// ---- VISUs/Parameter/Recipe/MOffset_1.TcVIS
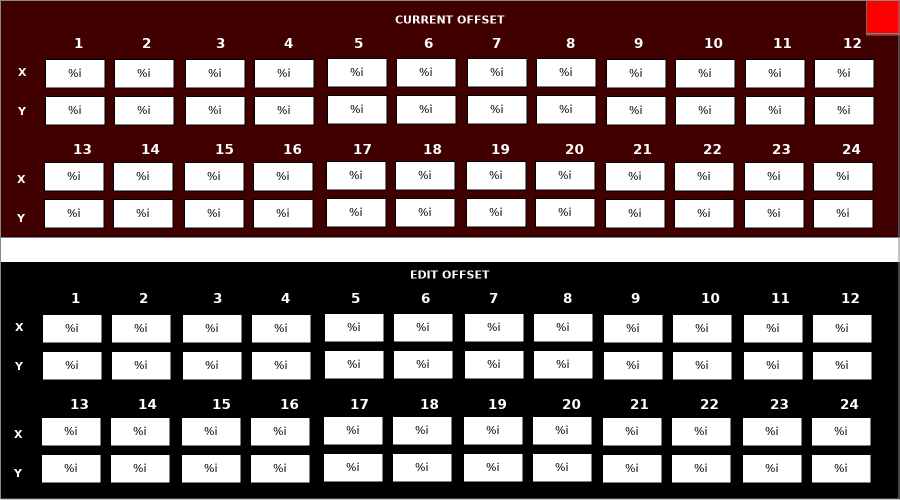
VISUALIZATION MOffset_1  // 900x500
    RoundedRectangle (0,0 900x237)
    Label (0,0 900x40), "CURRENT OFFSET"
    Label (15,55 25x35), "X"
    RoundedRectangle (45,59 60x29), "%i", text variable: Status_GVL.RecipeLine[1].OffsetPattern.Offset_X[1]
    Label (71,26 25x35), "1"
    RoundedRectangle (114,59 60x29), "%i", text variable: Status_GVL.RecipeLine[1].OffsetPattern.Offset_X[2]
    Label (139,26 25x35), "2"
    RoundedRectangle (185,59 60x29), "%i", text variable: Status_GVL.RecipeLine[1].OffsetPattern.Offset_X[3]
    RoundedRectangle (254,59 60x29), "%i", text variable: Status_GVL.RecipeLine[1].OffsetPattern.Offset_X[4]
    Label (15,94 25x35), "Y"
    RoundedRectangle (327,58 60x29), "%i", text variable: Status_GVL.RecipeLine[1].OffsetPattern.Offset_X[5]
    RoundedRectangle (396,58 60x29), "%i", text variable: Status_GVL.RecipeLine[1].OffsetPattern.Offset_X[6]
    RoundedRectangle (467,58 60x29), "%i", text variable: Status_GVL.RecipeLine[1].OffsetPattern.Offset_X[7]
    RoundedRectangle (536,58 60x29), "%i", text variable: Status_GVL.RecipeLine[1].OffsetPattern.Offset_X[8]
    RoundedRectangle (606,59 60x29), "%i", text variable: Status_GVL.RecipeLine[1].OffsetPattern.Offset_X[9]
    RoundedRectangle (675,59 60x29), "%i", text variable: Status_GVL.RecipeLine[1].OffsetPattern.Offset_X[10]
    Label (213,26 25x35), "3"
    Label (281,26 25x35), "4"
    Label (351,26 25x35), "5"
    Label (421,26 25x35), "6"
    Label (489,26 25x35), "7"
    Label (563,26 25x35), "8"
    Label (631,26 25x35), "9"
    Label (701,26 25x35), "10"
    RoundedRectangle (45,96 60x29), "%i", text variable: Status_GVL.RecipeLine[1].OffsetPattern.Offset_Y[1]
    RoundedRectangle (114,96 60x29), "%i", text variable: Status_GVL.RecipeLine[1].OffsetPattern.Offset_Y[2]
    RoundedRectangle (185,96 60x29), "%i", text variable: Status_GVL.RecipeLine[1].OffsetPattern.Offset_Y[3]
    RoundedRectangle (254,96 60x29), "%i", text variable: Status_GVL.RecipeLine[1].OffsetPattern.Offset_Y[4]
    RoundedRectangle (327,95 60x29), "%i", text variable: Status_GVL.RecipeLine[1].OffsetPattern.Offset_Y[5]
    RoundedRectangle (396,95 60x29), "%i", text variable: Status_GVL.RecipeLine[1].OffsetPattern.Offset_Y[6]
    RoundedRectangle (467,95 60x29), "%i", text variable: Status_GVL.RecipeLine[1].OffsetPattern.Offset_Y[7]
    RoundedRectangle (536,95 60x29), "%i", text variable: Status_GVL.RecipeLine[1].OffsetPattern.Offset_Y[8]
    RoundedRectangle (606,96 60x29), "%i", text variable: Status_GVL.RecipeLine[1].OffsetPattern.Offset_Y[9]
    RoundedRectangle (675,96 60x29), "%i", text variable: Status_GVL.RecipeLine[1].OffsetPattern.Offset_Y[10]
    Label (14,162 25x35), "X"
    RoundedRectangle (44,162 60x29), "%i", text variable: Status_GVL.RecipeLine[1].OffsetPattern.Offset_X[13]
    RoundedRectangle (113,162 60x29), "%i", text variable: Status_GVL.RecipeLine[1].OffsetPattern.Offset_X[14]
    RoundedRectangle (184,162 60x29), "%i", text variable: Status_GVL.RecipeLine[1].OffsetPattern.Offset_X[15]
    RoundedRectangle (253,162 60x29), "%i", text variable: Status_GVL.RecipeLine[1].OffsetPattern.Offset_X[16]
    Label (14,201 25x35), "Y"
    RoundedRectangle (326,161 60x29), "%i", text variable: Status_GVL.RecipeLine[1].OffsetPattern.Offset_X[17]
    RoundedRectangle (395,161 60x29), "%i", text variable: Status_GVL.RecipeLine[1].OffsetPattern.Offset_X[18]
    RoundedRectangle (466,161 60x29), "%i", text variable: Status_GVL.RecipeLine[1].OffsetPattern.Offset_X[19]
    RoundedRectangle (535,161 60x29), "%i", text variable: Status_GVL.RecipeLine[1].OffsetPattern.Offset_X[20]
    RoundedRectangle (605,162 60x29), "%i", text variable: Status_GVL.RecipeLine[1].OffsetPattern.Offset_X[21]
    RoundedRectangle (674,162 60x29), "%i", text variable: Status_GVL.RecipeLine[1].OffsetPattern.Offset_X[22]
    RoundedRectangle (44,199 60x29), "%i", text variable: Status_GVL.RecipeLine[1].OffsetPattern.Offset_Y[13]
    RoundedRectangle (113,199 60x29), "%i", text variable: Status_GVL.RecipeLine[1].OffsetPattern.Offset_Y[14]
    RoundedRectangle (184,199 60x29), "%i", text variable: Status_GVL.RecipeLine[1].OffsetPattern.Offset_Y[15]
    RoundedRectangle (253,199 60x29), "%i", text variable: Status_GVL.RecipeLine[1].OffsetPattern.Offset_Y[16]
    RoundedRectangle (326,198 60x29), "%i", text variable: Status_GVL.RecipeLine[1].OffsetPattern.Offset_Y[17]
    RoundedRectangle (395,198 60x29), "%i", text variable: Status_GVL.RecipeLine[1].OffsetPattern.Offset_Y[18]
    RoundedRectangle (466,198 60x29), "%i", text variable: Status_GVL.RecipeLine[1].OffsetPattern.Offset_Y[19]
    RoundedRectangle (535,198 60x29), "%i", text variable: Status_GVL.RecipeLine[1].OffsetPattern.Offset_Y[20]
    RoundedRectangle (605,199 60x29), "%i", text variable: Status_GVL.RecipeLine[1].OffsetPattern.Offset_Y[21]
    RoundedRectangle (674,199 60x29), "%i", text variable: Status_GVL.RecipeLine[1].OffsetPattern.Offset_Y[22]
    Label (70,132 25x35), "13"
    Label (138,132 25x35), "14"
    Label (212,132 25x35), "15"
    Label (280,132 25x35), "16"
    Label (350,132 25x35), "17"
    Label (420,132 25x35), "18"
    Label (488,132 25x35), "19"
    Label (562,132 25x35), "20"
    Label (630,132 25x35), "21"
    Label (700,132 25x35), "22"
    RoundedRectangle (0,262 900x237)
    Label (0,255 900x40), "EDIT OFFSET"
    Label (12,310 25x35), "X"
    RoundedRectangle (42,314 60x29), "%i", text variable: HMI_GVL.arRecipeHMI[1].OffsetPattern.Offset_X[1], input disabled if: Status_GVL.StsEdit[1]
        OnMouseClick: write the text variable via Default
    Label (68,281 25x35), "1"
    RoundedRectangle (111,314 60x29), "%i", text variable: HMI_GVL.arRecipeHMI[1].OffsetPattern.Offset_X[2], input disabled if: Status_GVL.StsEdit[1]
        OnMouseClick: write the text variable via Default
    Label (136,281 25x35), "2"
    RoundedRectangle (182,314 60x29), "%i", text variable: HMI_GVL.arRecipeHMI[1].OffsetPattern.Offset_X[3], input disabled if: Status_GVL.StsEdit[1]
        OnMouseClick: write the text variable via Default
    RoundedRectangle (251,314 60x29), "%i", text variable: HMI_GVL.arRecipeHMI[1].OffsetPattern.Offset_X[4], input disabled if: Status_GVL.StsEdit[1]
        OnMouseClick: write the text variable via Default
    Label (12,349 25x35), "Y"
    RoundedRectangle (324,313 60x29), "%i", text variable: HMI_GVL.arRecipeHMI[1].OffsetPattern.Offset_X[5], input disabled if: Status_GVL.StsEdit[1]
        OnMouseClick: write the text variable via Default
    RoundedRectangle (393,313 60x29), "%i", text variable: HMI_GVL.arRecipeHMI[1].OffsetPattern.Offset_X[6], input disabled if: Status_GVL.StsEdit[1]
        OnMouseClick: write the text variable via Default
    RoundedRectangle (464,313 60x29), "%i", text variable: HMI_GVL.arRecipeHMI[1].OffsetPattern.Offset_X[7], input disabled if: Status_GVL.StsEdit[1]
        OnMouseClick: write the text variable via Default
    RoundedRectangle (533,313 60x29), "%i", text variable: HMI_GVL.arRecipeHMI[1].OffsetPattern.Offset_X[8], input disabled if: Status_GVL.StsEdit[1]
        OnMouseClick: write the text variable via Default
    RoundedRectangle (603,314 60x29), "%i", text variable: HMI_GVL.arRecipeHMI[1].OffsetPattern.Offset_X[9], input disabled if: Status_GVL.StsEdit[1]
        OnMouseClick: write the text variable via Default
    RoundedRectangle (672,314 60x29), "%i", text variable: HMI_GVL.arRecipeHMI[1].OffsetPattern.Offset_X[10], input disabled if: Status_GVL.StsEdit[1]
        OnMouseClick: write the text variable via Default
    Label (210,281 25x35), "3"
    Label (278,281 25x35), "4"
    Label (348,281 25x35), "5"
    Label (418,281 25x35), "6"
    Label (486,281 25x35), "7"
    Label (560,281 25x35), "8"
    Label (628,281 25x35), "9"
    Label (698,281 25x35), "10"
    RoundedRectangle (42,351 60x29), "%i", text variable: HMI_GVL.arRecipeHMI[1].OffsetPattern.Offset_Y[1], input disabled if: Status_GVL.StsEdit[1]
        OnMouseClick: write the text variable via Default
    RoundedRectangle (111,351 60x29), "%i", text variable: HMI_GVL.arRecipeHMI[1].OffsetPattern.Offset_Y[2], input disabled if: Status_GVL.StsEdit[1]
        OnMouseClick: write the text variable via Default
    RoundedRectangle (182,351 60x29), "%i", text variable: HMI_GVL.arRecipeHMI[1].OffsetPattern.Offset_Y[3], input disabled if: Status_GVL.StsEdit[1]
        OnMouseClick: write the text variable via Default
    RoundedRectangle (251,351 60x29), "%i", text variable: HMI_GVL.arRecipeHMI[1].OffsetPattern.Offset_Y[4], input disabled if: Status_GVL.StsEdit[1]
        OnMouseClick: write the text variable via Default
    RoundedRectangle (324,350 60x29), "%i", text variable: HMI_GVL.arRecipeHMI[1].OffsetPattern.Offset_Y[5], input disabled if: Status_GVL.StsEdit[1]
        OnMouseClick: write the text variable via Default
    RoundedRectangle (393,350 60x29), "%i", text variable: HMI_GVL.arRecipeHMI[1].OffsetPattern.Offset_Y[6], input disabled if: Status_GVL.StsEdit[1]
        OnMouseClick: write the text variable via Default
    RoundedRectangle (464,350 60x29), "%i", text variable: HMI_GVL.arRecipeHMI[1].OffsetPattern.Offset_Y[7], input disabled if: Status_GVL.StsEdit[1]
        OnMouseClick: write the text variable via Default
    RoundedRectangle (533,350 60x29), "%i", text variable: HMI_GVL.arRecipeHMI[1].OffsetPattern.Offset_Y[8], input disabled if: Status_GVL.StsEdit[1]
        OnMouseClick: write the text variable via Default
    RoundedRectangle (603,351 60x29), "%i", text variable: HMI_GVL.arRecipeHMI[1].OffsetPattern.Offset_Y[9], input disabled if: Status_GVL.StsEdit[1]
        OnMouseClick: write the text variable via Default
    RoundedRectangle (672,351 60x29), "%i", text variable: HMI_GVL.arRecipeHMI[1].OffsetPattern.Offset_Y[10], input disabled if: Status_GVL.StsEdit[1]
        OnMouseClick: write the text variable via Default
    Label (11,417 25x35), "X"
    RoundedRectangle (41,417 60x29), "%i", text variable: HMI_GVL.arRecipeHMI[1].OffsetPattern.Offset_X[13], input disabled if: Status_GVL.StsEdit[1]
        OnMouseClick: write the text variable via Default
    RoundedRectangle (110,417 60x29), "%i", text variable: HMI_GVL.arRecipeHMI[1].OffsetPattern.Offset_X[14], input disabled if: Status_GVL.StsEdit[1]
        OnMouseClick: write the text variable via Default
    RoundedRectangle (181,417 60x29), "%i", text variable: HMI_GVL.arRecipeHMI[1].OffsetPattern.Offset_X[15], input disabled if: Status_GVL.StsEdit[1]
        OnMouseClick: write the text variable via Default
    RoundedRectangle (250,417 60x29), "%i", text variable: HMI_GVL.arRecipeHMI[1].OffsetPattern.Offset_X[16], input disabled if: Status_GVL.StsEdit[1]
        OnMouseClick: write the text variable via Default
    Label (11,456 25x35), "Y"
    RoundedRectangle (323,416 60x29), "%i", text variable: HMI_GVL.arRecipeHMI[1].OffsetPattern.Offset_X[17], input disabled if: Status_GVL.StsEdit[1]
        OnMouseClick: write the text variable via Default
    RoundedRectangle (392,416 60x29), "%i", text variable: HMI_GVL.arRecipeHMI[1].OffsetPattern.Offset_X[18], input disabled if: Status_GVL.StsEdit[1]
        OnMouseClick: write the text variable via Default
    RoundedRectangle (463,416 60x29), "%i", text variable: HMI_GVL.arRecipeHMI[1].OffsetPattern.Offset_X[19], input disabled if: Status_GVL.StsEdit[1]
        OnMouseClick: write the text variable via Default
    RoundedRectangle (532,416 60x29), "%i", text variable: HMI_GVL.arRecipeHMI[1].OffsetPattern.Offset_X[20], input disabled if: Status_GVL.StsEdit[1]
        OnMouseClick: write the text variable via Default
    RoundedRectangle (602,417 60x29), "%i", text variable: HMI_GVL.arRecipeHMI[1].OffsetPattern.Offset_X[21], input disabled if: Status_GVL.StsEdit[1]
        OnMouseClick: write the text variable via Default
    RoundedRectangle (671,417 60x29), "%i", text variable: HMI_GVL.arRecipeHMI[1].OffsetPattern.Offset_X[22], input disabled if: Status_GVL.StsEdit[1]
        OnMouseClick: write the text variable via Default
    RoundedRectangle (41,454 60x29), "%i", text variable: HMI_GVL.arRecipeHMI[1].OffsetPattern.Offset_Y[13], input disabled if: Status_GVL.StsEdit[1]
        OnMouseClick: write the text variable via Default
    RoundedRectangle (110,454 60x29), "%i", text variable: HMI_GVL.arRecipeHMI[1].OffsetPattern.Offset_Y[14], input disabled if: Status_GVL.StsEdit[1]
        OnMouseClick: write the text variable via Default
    RoundedRectangle (181,454 60x29), "%i", text variable: HMI_GVL.arRecipeHMI[1].OffsetPattern.Offset_Y[15], input disabled if: Status_GVL.StsEdit[1]
        OnMouseClick: write the text variable via Default
    RoundedRectangle (250,454 60x29), "%i", text variable: HMI_GVL.arRecipeHMI[1].OffsetPattern.Offset_Y[16], input disabled if: Status_GVL.StsEdit[1]
        OnMouseClick: write the text variable via Default
    RoundedRectangle (323,453 60x29), "%i", text variable: HMI_GVL.arRecipeHMI[1].OffsetPattern.Offset_Y[17], input disabled if: Status_GVL.StsEdit[1]
        OnMouseClick: write the text variable via Default
    RoundedRectangle (392,453 60x29), "%i", text variable: HMI_GVL.arRecipeHMI[1].OffsetPattern.Offset_Y[18], input disabled if: Status_GVL.StsEdit[1]
        OnMouseClick: write the text variable via Default
    RoundedRectangle (463,453 60x29), "%i", text variable: HMI_GVL.arRecipeHMI[1].OffsetPattern.Offset_Y[19], input disabled if: Status_GVL.StsEdit[1]
        OnMouseClick: write the text variable via Default
    RoundedRectangle (532,453 60x29), "%i", text variable: HMI_GVL.arRecipeHMI[1].OffsetPattern.Offset_Y[20], input disabled if: Status_GVL.StsEdit[1]
        OnMouseClick: write the text variable via Default
    RoundedRectangle (602,454 60x29), "%i", text variable: HMI_GVL.arRecipeHMI[1].OffsetPattern.Offset_Y[21], input disabled if: Status_GVL.StsEdit[1]
        OnMouseClick: write the text variable via Default
    RoundedRectangle (671,454 60x29), "%i", text variable: HMI_GVL.arRecipeHMI[1].OffsetPattern.Offset_Y[22], input disabled if: Status_GVL.StsEdit[1]
        OnMouseClick: write the text variable via Default
    Label (67,387 25x35), "13"
    Label (135,387 25x35), "14"
    Label (209,387 25x35), "15"
    Label (277,387 25x35), "16"
    Label (347,387 25x35), "17"
    Label (417,387 25x35), "18"
    Label (485,387 25x35), "19"
    Label (559,387 25x35), "20"
    Label (627,387 25x35), "21"
    Label (697,387 25x35), "22"
    Button (866,0 35x35), image: VisuSymbols.Symbols.Wrong
        OnMouseClick: CloseDialog Dialog=MOffset_1, Result=OK, NumpadKeypadSet=True
    RoundedRectangle (745,59 60x29), "%i", text variable: Status_GVL.RecipeLine[1].OffsetPattern.Offset_X[11]
    RoundedRectangle (814,59 60x29), "%i", text variable: Status_GVL.RecipeLine[1].OffsetPattern.Offset_X[12]
    Label (770,26 25x35), "11"
    Label (840,26 25x35), "12"
    RoundedRectangle (745,96 60x29), "%i", text variable: Status_GVL.RecipeLine[1].OffsetPattern.Offset_Y[11]
    RoundedRectangle (814,96 60x29), "%i", text variable: Status_GVL.RecipeLine[1].OffsetPattern.Offset_Y[12]
    RoundedRectangle (744,162 60x29), "%i", text variable: Status_GVL.RecipeLine[1].OffsetPattern.Offset_X[23]
    RoundedRectangle (813,162 60x29), "%i", text variable: Status_GVL.RecipeLine[1].OffsetPattern.Offset_X[24]
    RoundedRectangle (744,199 60x29), "%i", text variable: Status_GVL.RecipeLine[1].OffsetPattern.Offset_Y[23]
    RoundedRectangle (813,199 60x29), "%i", text variable: Status_GVL.RecipeLine[1].OffsetPattern.Offset_Y[24]
    Label (769,132 25x35), "23"
    Label (839,132 25x35), "24"
    RoundedRectangle (743,314 60x29), "%i", text variable: HMI_GVL.arRecipeHMI[1].OffsetPattern.Offset_X[11], input disabled if: Status_GVL.StsEdit[1]
        OnMouseClick: write the text variable via Default
    RoundedRectangle (812,314 60x29), "%i", text variable: HMI_GVL.arRecipeHMI[1].OffsetPattern.Offset_X[12], input disabled if: Status_GVL.StsEdit[1]
        OnMouseClick: write the text variable via Default
    Label (768,281 25x35), "11"
    Label (838,281 25x35), "12"
    RoundedRectangle (743,351 60x29), "%i", text variable: HMI_GVL.arRecipeHMI[1].OffsetPattern.Offset_Y[11], input disabled if: Status_GVL.StsEdit[1]
        OnMouseClick: write the text variable via Default
    RoundedRectangle (812,351 60x29), "%i", text variable: HMI_GVL.arRecipeHMI[1].OffsetPattern.Offset_Y[12], input disabled if: Status_GVL.StsEdit[1]
        OnMouseClick: write the text variable via Default
    RoundedRectangle (742,417 60x29), "%i", text variable: HMI_GVL.arRecipeHMI[1].OffsetPattern.Offset_X[23], input disabled if: Status_GVL.StsEdit[1]
        OnMouseClick: write the text variable via Default
    RoundedRectangle (811,417 60x29), "%i", text variable: HMI_GVL.arRecipeHMI[1].OffsetPattern.Offset_X[24], input disabled if: Status_GVL.StsEdit[1]
        OnMouseClick: write the text variable via Default
    RoundedRectangle (742,454 60x29), "%i", text variable: HMI_GVL.arRecipeHMI[1].OffsetPattern.Offset_Y[23], input disabled if: Status_GVL.StsEdit[1]
        OnMouseClick: write the text variable via Default
    RoundedRectangle (811,454 60x29), "%i", text variable: HMI_GVL.arRecipeHMI[1].OffsetPattern.Offset_Y[24], input disabled if: Status_GVL.StsEdit[1]
        OnMouseClick: write the text variable via Default
    Label (767,387 25x35), "23"
    Label (837,387 25x35), "24"
END_VISUALIZATION

// ---- VISUs/Parameter/Recipe/MRecipe_2.TcVIS
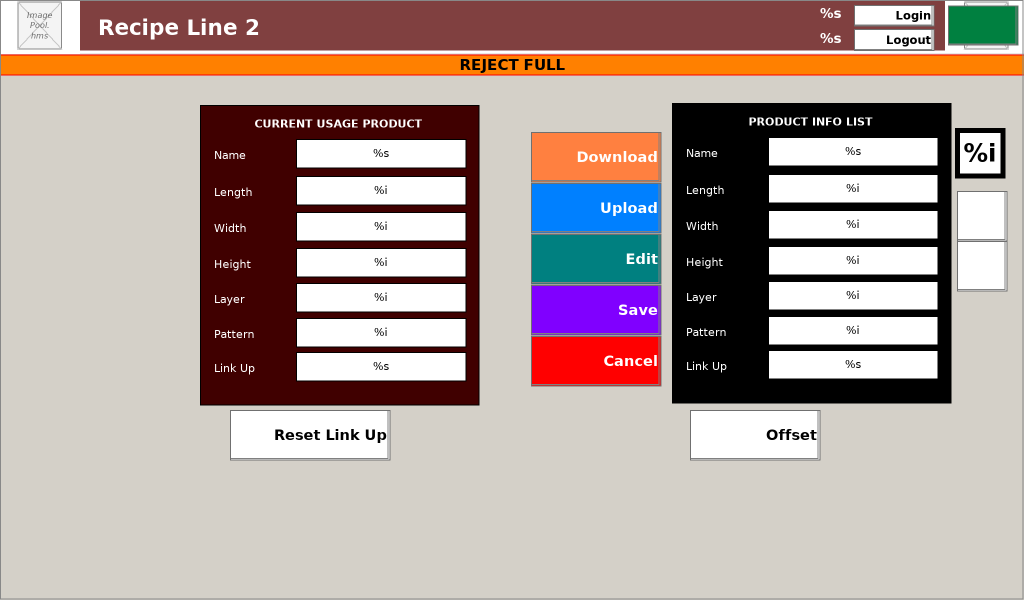
VISUALIZATION MRecipe_2  // 1024x600
    Frame (0,-2 1021x55)
        shows Header()
    Label (95,15 250x25), "Recipe Line 2"
    RoundedRectangle (672,103 279x300)
    Label (697,102 227x40), "PRODUCT INFO LIST"
    Label (683,136 78x35), "Name"
    RoundedRectangle (768,137 170x29), "%s", text variable: HMI_GVL.arRecipeHMI[2].ProductName, input disabled if: Status_GVL.StsEdit[2]
        OnMouseClick: write the text variable via Default
    Label (683,173 78x35), "Length"
    RoundedRectangle (768,174 170x29), "%i", text variable: HMI_GVL.arRecipeHMI[2].ProductLength, input disabled if: Status_GVL.StsEdit[2]
        OnMouseClick: write the text variable via Default
    Label (683,209 78x35), "Width"
    RoundedRectangle (768,210 170x29), "%i", text variable: HMI_GVL.arRecipeHMI[2].ProductWidth, input disabled if: Status_GVL.StsEdit[2]
        OnMouseClick: write the text variable via Default
    Label (683,245 78x35), "Height"
    RoundedRectangle (768,246 170x29), "%i", text variable: HMI_GVL.arRecipeHMI[2].ProductHeight, input disabled if: Status_GVL.StsEdit[2]
        OnMouseClick: write the text variable via Default
    Label (683,280 78x35), "Layer"
    RoundedRectangle (768,281 170x29), "%i", text variable: HMI_GVL.arRecipeHMI[2].Stacking, input disabled if: Status_GVL.StsEdit[2]
        OnMouseClick: write the text variable via Default
    Label (683,315 78x35), "Pattern"
    RoundedRectangle (768,316 170x29), "%i", text variable: HMI_GVL.arRecipeHMI[2].ProductPattern, input disabled if: Status_GVL.StsEdit[2]
        OnMouseClick: write the text variable via Default
    Label (683,349 78x35), "Link Up"
    RoundedRectangle (768,350 170x29), "%s", text variable: HMI_GVL.arRecipeHMI[2].LinkUpSource, input disabled if: Status_GVL.StsEdit[2]
        OnMouseClick: write the text variable via Default
    Button (531,132 130x50), "Download", image: VisuSymbols.Symbols.Download
        tap Status_GVL.Download[2]
    Button (531,183 130x50), "Upload", image: VisuSymbols.Symbols.Eject
        tap Status_GVL.Upload[2]
    Button (531,234 130x50), "Edit", image: VisuSymbols.Symbols.Edit
        tap Status_GVL.Edit[2]
    Button (531,285 130x50), "Save", invisible if: Status_GVL.StsEdit[2], image: VisuSymbols.Symbols.Save
        tap Status_GVL.Save[2]
    Button (531,336 130x50), "Cancel", invisible if: Status_GVL.StsEdit[2], image: VisuSymbols.Symbols.Wrong
        tap Status_GVL.Cancel[2]
    RoundedRectangle (955,128 50x50), "%i", text variable: Status_GVL.RecipeNumber[2]
        OnMouseClick: write the text variable via Default
    Button (957,191 50x50), image: VisuSymbols.Symbols.TriangleUp
        OnMouseClick: execute {
            IF Status_GVL.StsEdit[2] THEN
            Status_GVL.RecipeNumber[2] := Status_GVL.RecipeNumber[2]+1;
            END_IF
        }
    Button (957,241 50x50), image: VisuSymbols.Symbols.TriangleDown
        OnMouseClick: execute {
            IF Status_GVL.StsEdit[2] THEN
            Status_GVL.RecipeNumber[2] := Status_GVL.RecipeNumber[2]-1;
            END_IF
        }
    Button (690,410 130x50), "Offset", image: VisuSymbols.Symbols.Centered
        OnMouseClick: OpenDialog Dialog=MOffset_2, OpenModal=True, OpenCentered=True, PositionY=0
    Group (200,104 279x356)
        RoundedRectangle (0,1 279x300)
        Label (25,0 227x40), "CURRENT USAGE PRODUCT"
        Label (11,34 78x35), "Name"
        RoundedRectangle (96,35 170x29), "%s", text variable: Status_GVL.RecipeLine[2].ProductName
        Label (11,71 78x35), "Length"
        RoundedRectangle (96,72 170x29), "%i", text variable: Status_GVL.RecipeLine[2].ProductLength
        Label (11,107 78x35), "Width"
        RoundedRectangle (96,108 170x29), "%i", text variable: Status_GVL.RecipeLine[2].ProductWidth
        Label (11,143 78x35), "Height"
        RoundedRectangle (96,144 170x29), "%i", text variable: Status_GVL.RecipeLine[2].ProductHeight
        Label (11,178 78x35), "Layer"
        RoundedRectangle (96,179 170x29), "%i", text variable: Status_GVL.RecipeLine[2].Stacking
        Label (11,213 78x35), "Pattern"
        RoundedRectangle (96,214 170x29), "%i", text variable: Status_GVL.RecipeLine[2].ProductPattern
        Label (11,247 78x35), "Link Up"
        RoundedRectangle (96,248 170x29), "%s", text variable: Status_GVL.RecipeLine[2].LinkUpSource
        Button (30,306 160x50), "Reset Link Up", image: VisuSymbols.Symbols.Eraser
            tap HMI_GVL.Reset_LinkUp[2]
END_VISUALIZATION

// ---- VISUs/Parameter/Recipe/MRecipe_3.TcVIS
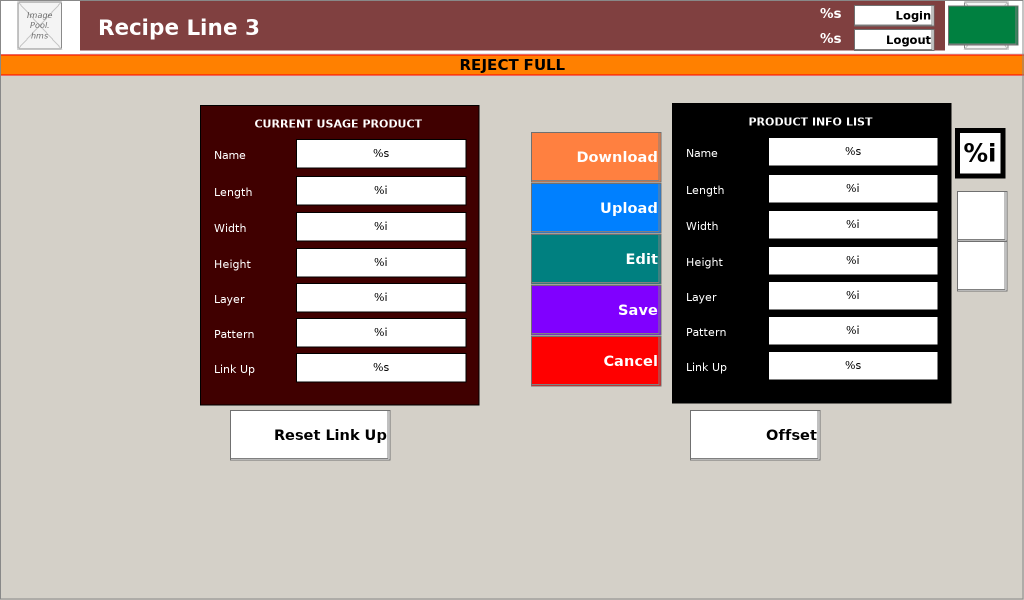
VISUALIZATION MRecipe_3  // 1024x600
    Frame (0,-2 1021x55)
        shows Header()
    Label (95,15 250x25), "Recipe Line 3"
    RoundedRectangle (672,103 279x300)
    Label (697,102 227x40), "PRODUCT INFO LIST"
    Label (683,136 78x35), "Name"
    RoundedRectangle (768,137 170x29), "%s", text variable: HMI_GVL.arRecipeHMI[3].ProductName, input disabled if: Status_GVL.StsEdit[3]
        OnMouseClick: write the text variable via Default
    Label (683,173 78x35), "Length"
    RoundedRectangle (768,174 170x29), "%i", text variable: HMI_GVL.arRecipeHMI[3].ProductLength, input disabled if: Status_GVL.StsEdit[3]
        OnMouseClick: write the text variable via Default
    Label (683,209 78x35), "Width"
    RoundedRectangle (768,210 170x29), "%i", text variable: HMI_GVL.arRecipeHMI[3].ProductWidth, input disabled if: Status_GVL.StsEdit[3]
        OnMouseClick: write the text variable via Default
    Label (683,245 78x35), "Height"
    RoundedRectangle (768,246 170x29), "%i", text variable: HMI_GVL.arRecipeHMI[3].ProductHeight, input disabled if: Status_GVL.StsEdit[3]
        OnMouseClick: write the text variable via Default
    Label (683,280 78x35), "Layer"
    RoundedRectangle (768,281 170x29), "%i", text variable: HMI_GVL.arRecipeHMI[3].Stacking, input disabled if: Status_GVL.StsEdit[3]
        OnMouseClick: write the text variable via Default
    Label (683,315 78x35), "Pattern"
    RoundedRectangle (768,316 170x29), "%i", text variable: HMI_GVL.arRecipeHMI[3].ProductPattern, input disabled if: Status_GVL.StsEdit[3]
        OnMouseClick: write the text variable via Default
    Label (683,350 78x35), "Link Up"
    RoundedRectangle (768,351 170x29), "%s", text variable: HMI_GVL.arRecipeHMI[3].LinkUpSource, input disabled if: Status_GVL.StsEdit[3]
        OnMouseClick: write the text variable via Default
    Button (531,132 130x50), "Download", image: VisuSymbols.Symbols.Download
        tap Status_GVL.Download[3]
    Button (531,183 130x50), "Upload", image: VisuSymbols.Symbols.Eject
        tap Status_GVL.Upload[3]
    Button (531,234 130x50), "Edit", image: VisuSymbols.Symbols.Edit
        tap Status_GVL.Edit[3]
    Button (531,285 130x50), "Save", invisible if: Status_GVL.StsEdit[3], image: VisuSymbols.Symbols.Save
        tap Status_GVL.Save[3]
    Button (531,336 130x50), "Cancel", invisible if: Status_GVL.StsEdit[3], image: VisuSymbols.Symbols.Wrong
        tap Status_GVL.Cancel[3]
    RoundedRectangle (955,128 50x50), "%i", text variable: Status_GVL.RecipeNumber[3]
        OnMouseClick: write the text variable via Default
    Button (957,191 50x50), image: VisuSymbols.Symbols.TriangleUp
        OnMouseClick: execute {
            IF Status_GVL.StsEdit[3] THEN
            Status_GVL.RecipeNumber[3] := Status_GVL.RecipeNumber[3]+1;
            END_IF
        }
    Button (957,241 50x50), image: VisuSymbols.Symbols.TriangleDown
        OnMouseClick: execute {
            IF Status_GVL.StsEdit[3] THEN
            Status_GVL.RecipeNumber[3] := Status_GVL.RecipeNumber[3]-1;
            END_IF
        }
    Button (690,410 130x50), "Offset", image: VisuSymbols.Symbols.Centered
        OnMouseClick: OpenDialog Dialog=MOffset_3, OpenModal=True, OpenCentered=True, PositionY=0
    Group (200,104 279x356)
        RoundedRectangle (0,1 279x300)
        Label (25,0 227x40), "CURRENT USAGE PRODUCT"
        Label (11,34 78x35), "Name"
        RoundedRectangle (96,35 170x29), "%s", text variable: Status_GVL.RecipeLine[3].ProductName
        Label (11,71 78x35), "Length"
        RoundedRectangle (96,72 170x29), "%i", text variable: Status_GVL.RecipeLine[3].ProductLength
        Label (11,107 78x35), "Width"
        RoundedRectangle (96,108 170x29), "%i", text variable: Status_GVL.RecipeLine[3].ProductWidth
        Label (11,143 78x35), "Height"
        RoundedRectangle (96,144 170x29), "%i", text variable: Status_GVL.RecipeLine[3].ProductHeight
        Label (11,178 78x35), "Layer"
        RoundedRectangle (96,179 170x29), "%i", text variable: Status_GVL.RecipeLine[3].Stacking
        Label (11,213 78x35), "Pattern"
        RoundedRectangle (96,214 170x29), "%i", text variable: Status_GVL.RecipeLine[3].ProductPattern
        Label (11,248 78x35), "Link Up"
        RoundedRectangle (96,249 170x29), "%s", text variable: Status_GVL.RecipeLine[3].LinkUpSource
        Button (30,306 160x50), "Reset Link Up", image: VisuSymbols.Symbols.Eraser
            tap HMI_GVL.Reset_LinkUp[3]
END_VISUALIZATION

// ---- VISUs/Parameter/Recipe/MRecipe_4.TcVIS
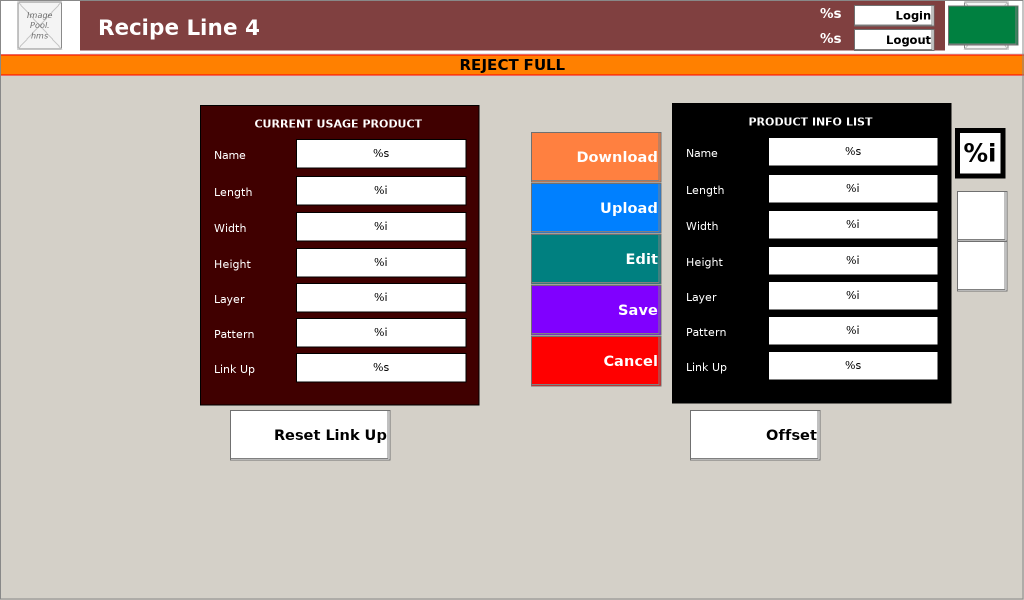
VISUALIZATION MRecipe_4  // 1024x600
    Frame (0,-2 1021x55)
        shows Header()
    Label (95,15 250x25), "Recipe Line 4"
    RoundedRectangle (672,103 279x300)
    Label (697,102 227x40), "PRODUCT INFO LIST"
    Label (683,136 78x35), "Name"
    RoundedRectangle (768,137 170x29), "%s", text variable: HMI_GVL.arRecipeHMI[4].ProductName, input disabled if: Status_GVL.StsEdit[4]
        OnMouseClick: write the text variable via Default
    Label (683,173 78x35), "Length"
    RoundedRectangle (768,174 170x29), "%i", text variable: HMI_GVL.arRecipeHMI[4].ProductLength, input disabled if: Status_GVL.StsEdit[4]
        OnMouseClick: write the text variable via Default
    Label (683,209 78x35), "Width"
    RoundedRectangle (768,210 170x29), "%i", text variable: HMI_GVL.arRecipeHMI[4].ProductWidth, input disabled if: Status_GVL.StsEdit[4]
        OnMouseClick: write the text variable via Default
    Label (683,245 78x35), "Height"
    RoundedRectangle (768,246 170x29), "%i", text variable: HMI_GVL.arRecipeHMI[4].ProductHeight, input disabled if: Status_GVL.StsEdit[4]
        OnMouseClick: write the text variable via Default
    Label (683,280 78x35), "Layer"
    RoundedRectangle (768,281 170x29), "%i", text variable: HMI_GVL.arRecipeHMI[4].Stacking, input disabled if: Status_GVL.StsEdit[4]
        OnMouseClick: write the text variable via Default
    Label (683,315 78x35), "Pattern"
    RoundedRectangle (768,316 170x29), "%i", text variable: HMI_GVL.arRecipeHMI[4].ProductPattern, input disabled if: Status_GVL.StsEdit[4]
        OnMouseClick: write the text variable via Default
    Label (683,350 78x35), "Link Up"
    RoundedRectangle (768,351 170x29), "%s", text variable: HMI_GVL.arRecipeHMI[4].LinkUpSource, input disabled if: Status_GVL.StsEdit[4]
        OnMouseClick: write the text variable via Default
    Button (531,132 130x50), "Download", image: VisuSymbols.Symbols.Download
        tap Status_GVL.Download[4]
    Button (531,183 130x50), "Upload", image: VisuSymbols.Symbols.Eject
        tap Status_GVL.Upload[4]
    Button (531,234 130x50), "Edit", image: VisuSymbols.Symbols.Edit
        tap Status_GVL.Edit[4]
    Button (531,285 130x50), "Save", invisible if: Status_GVL.StsEdit[4], image: VisuSymbols.Symbols.Save
        tap Status_GVL.Save[4]
    Button (531,336 130x50), "Cancel", invisible if: Status_GVL.StsEdit[4], image: VisuSymbols.Symbols.Wrong
        tap Status_GVL.Cancel[4]
    RoundedRectangle (955,128 50x50), "%i", text variable: Status_GVL.RecipeNumber[4]
        OnMouseClick: write the text variable via Default
    Button (957,191 50x50), image: VisuSymbols.Symbols.TriangleUp
        OnMouseClick: execute {
            IF Status_GVL.StsEdit[4] THEN
            Status_GVL.RecipeNumber[4] := Status_GVL.RecipeNumber[4]+1;
            END_IF
        }
    Button (957,241 50x50), image: VisuSymbols.Symbols.TriangleDown
        OnMouseClick: execute {
            IF Status_GVL.StsEdit[4] THEN
            Status_GVL.RecipeNumber[4] := Status_GVL.RecipeNumber[4]-1;
            END_IF
        }
    Button (690,410 130x50), "Offset", image: VisuSymbols.Symbols.Centered
        OnMouseClick: OpenDialog Dialog=MOffset_4, OpenModal=True, OpenCentered=True, PositionY=0
    Group (200,104 279x356)
        RoundedRectangle (0,1 279x300)
        Label (25,0 227x40), "CURRENT USAGE PRODUCT"
        Label (11,34 78x35), "Name"
        RoundedRectangle (96,35 170x29), "%s", text variable: Status_GVL.RecipeLine[4].ProductName
        Label (11,71 78x35), "Length"
        RoundedRectangle (96,72 170x29), "%i", text variable: Status_GVL.RecipeLine[4].ProductLength
        Label (11,107 78x35), "Width"
        RoundedRectangle (96,108 170x29), "%i", text variable: Status_GVL.RecipeLine[4].ProductWidth
        Label (11,143 78x35), "Height"
        RoundedRectangle (96,144 170x29), "%i", text variable: Status_GVL.RecipeLine[4].ProductHeight
        Label (11,178 78x35), "Layer"
        RoundedRectangle (96,179 170x29), "%i", text variable: Status_GVL.RecipeLine[4].Stacking
        Label (11,213 78x35), "Pattern"
        RoundedRectangle (96,214 170x29), "%i", text variable: Status_GVL.RecipeLine[4].ProductPattern
        Label (11,248 78x35), "Link Up"
        RoundedRectangle (96,249 170x29), "%s", text variable: Status_GVL.RecipeLine[4].LinkUpSource
        Button (30,306 160x50), "Reset Link Up", image: VisuSymbols.Symbols.Eraser
            tap HMI_GVL.Reset_LinkUp[4]
END_VISUALIZATION

// ---- VISUs/PLC Status/P1 - Panel Robot/P1_DI1.TcVIS
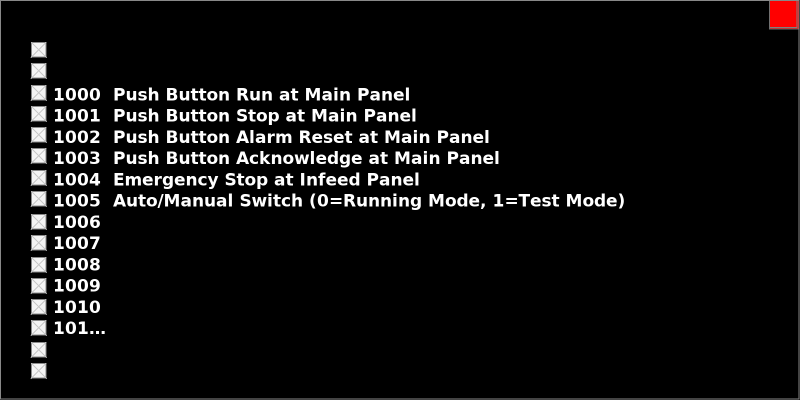
VISUALIZATION P1_DI1  // 800x400, background image 
    ImageSwitcher (31,42 15x15), variable: InputOutput_GVL.xIn1000, behaviour: TOGGLE
    Label (50,16 625x391), "1000 Push Button Run at Main Panel 1001 Push Button Stop at Main Panel 1002 Push Button Alarm Reset at Main Panel 1003 Push Button Acknowledge at Main Panel 1004 Emergency Stop at Infeed Panel 1005 Auto/Manual Switch (0=Running Mode, 1=Test Mode) 1006 1007 1008 1009 1010 1011 1012 1013 1014 1015 Pressure Switch for Main Panel"
    ImageSwitcher (31,63 15x15), variable: InputOutput_GVL.xIn1001, behaviour: TOGGLE
    ImageSwitcher (31,85 15x15), variable: InputOutput_GVL.xIn1002, behaviour: TOGGLE
    ImageSwitcher (31,106 15x15), variable: InputOutput_GVL.xIn1003, behaviour: TOGGLE
    ImageSwitcher (31,127 15x15), variable: InputOutput_GVL.xIn1004, behaviour: TOGGLE
    ImageSwitcher (31,148 15x15), variable: InputOutput_GVL.xIn1005, behaviour: TOGGLE
    ImageSwitcher (31,170 15x15), variable: InputOutput_GVL.xIn1006, behaviour: TOGGLE
    ImageSwitcher (31,191 15x15), variable: InputOutput_GVL.xIn1007, behaviour: TOGGLE
    ImageSwitcher (31,214 15x15), variable: InputOutput_GVL.xIn1008, behaviour: TOGGLE
    ImageSwitcher (31,235 15x15), variable: InputOutput_GVL.xIn1009, behaviour: TOGGLE
    ImageSwitcher (31,257 15x15), variable: InputOutput_GVL.xIn1010, behaviour: TOGGLE
    ImageSwitcher (31,278 15x15), variable: InputOutput_GVL.xIn1011, behaviour: TOGGLE
    ImageSwitcher (31,299 15x15), variable: InputOutput_GVL.xIn1012, behaviour: TOGGLE
    ImageSwitcher (31,320 15x15), variable: InputOutput_GVL.xIn1013, behaviour: TOGGLE
    ImageSwitcher (31,342 15x15), variable: InputOutput_GVL.xIn1014, behaviour: TOGGLE
    ImageSwitcher (31,363 15x15), variable: InputOutput_GVL.xIn1015, behaviour: TOGGLE
    Button (769,-1 30x30), image: VisuSymbols.Symbols.Wrong
        OnMouseClick: CloseDialog Dialog=P1_DI1, Result=OK, NumpadKeypadSet=True
END_VISUALIZATION

// ---- VISUs/PLC Status/P1 - Panel Robot/P1_DI2.TcVIS
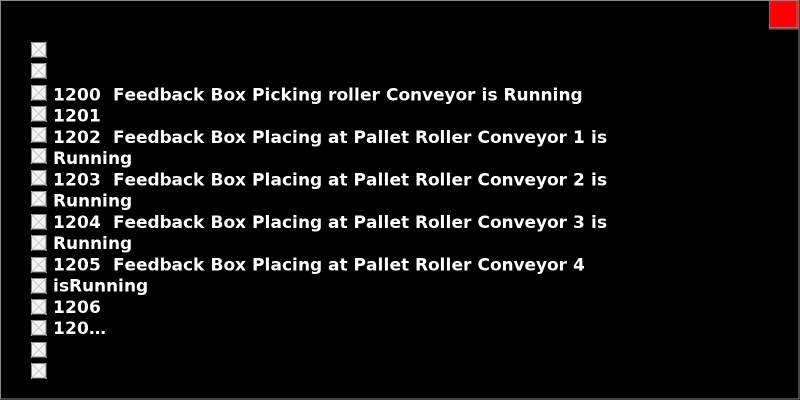
VISUALIZATION P1_DI2  // 800x400, background image 
    ImageSwitcher (31,42 15x15), variable: InputOutput_GVL.xIn1200, behaviour: TOGGLE
    Label (50,16 625x391), "1200 Feedback Box Picking roller Conveyor is Running 1201 1202 Feedback Box Placing at Pallet Roller Conveyor 1 is Running 1203 Feedback Box Placing at Pallet Roller Conveyor 2 is Running 1204 Feedback Box Placing at Pallet Roller Conveyor 3 is Running 1205 Feedback Box Placing at Pallet Roller Conveyor 4 isRunning 1206 1207 1208 1209 1210 1211 RSW Pneumatic Box Centring When Rtc 1212 RSW Pneumatic Gap Maker When Adv 1213 RSW Pneumatic Gap Maker When Rtc 1214 RSW Pneumatic Stopper Transfer When Rtc 1215"
    ImageSwitcher (31,63 15x15), variable: InputOutput_GVL.xIn1201, behaviour: TOGGLE
    ImageSwitcher (31,85 15x15), variable: InputOutput_GVL.xIn1202, behaviour: TOGGLE
    ImageSwitcher (31,106 15x15), variable: InputOutput_GVL.xIn1203, behaviour: TOGGLE
    ImageSwitcher (31,127 15x15), variable: InputOutput_GVL.xIn1204, behaviour: TOGGLE
    ImageSwitcher (31,148 15x15), variable: InputOutput_GVL.xIn1205, behaviour: TOGGLE
    ImageSwitcher (31,170 15x15), variable: InputOutput_GVL.xIn1206, behaviour: TOGGLE
    ImageSwitcher (31,191 15x15), variable: InputOutput_GVL.xIn1207, behaviour: TOGGLE
    ImageSwitcher (31,214 15x15), variable: InputOutput_GVL.xIn1208, behaviour: TOGGLE
    ImageSwitcher (31,235 15x15), variable: InputOutput_GVL.xIn1209, behaviour: TOGGLE
    ImageSwitcher (31,257 15x15), variable: InputOutput_GVL.xIn1210, behaviour: TOGGLE
    ImageSwitcher (31,278 15x15), variable: InputOutput_GVL.xIn1211, behaviour: TOGGLE
    ImageSwitcher (31,299 15x15), variable: InputOutput_GVL.xIn1212, behaviour: TOGGLE
    ImageSwitcher (31,320 15x15), variable: InputOutput_GVL.xIn1213, behaviour: TOGGLE
    ImageSwitcher (31,342 15x15), variable: InputOutput_GVL.xIn1214, behaviour: TOGGLE
    ImageSwitcher (31,363 15x15), variable: InputOutput_GVL.xIn1215, behaviour: TOGGLE
    Button (769,-1 30x30), image: VisuSymbols.Symbols.Wrong
        OnMouseClick: CloseDialog Dialog=P1_DI2, Result=OK, NumpadKeypadSet=True
END_VISUALIZATION

// ---- VISUs/PLC Status/P1 - Panel Robot/P1_DI3.TcVIS
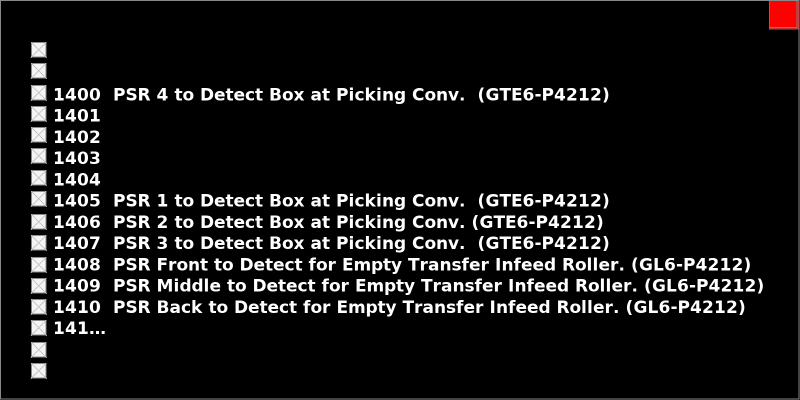
VISUALIZATION P1_DI3  // 800x400, background image 
    ImageSwitcher (31,42 15x15), variable: InputOutput_GVL.xIn1400, behaviour: TOGGLE
    Label (50,16 732x391), "1400 PSR 4 to Detect Box at Picking Conv. (GTE6-P4212) 1401 1402 1403 1404 1405 PSR 1 to Detect Box at Picking Conv. (GTE6-P4212) 1406 PSR 2 to Detect Box at Picking Conv. (GTE6-P4212) 1407 PSR 3 to Detect Box at Picking Conv. (GTE6-P4212) 1408 PSR Front to Detect for Empty Transfer Infeed Roller. (GL6-P4212) 1409 PSR Middle to Detect for Empty Transfer Infeed Roller. (GL6-P4212) 1410 PSR Back to Detect for Empty Transfer Infeed Roller. (GL6-P4212) 1411 1412 1413 1414 Request Release Solenoid Door Robot 1415 Feedback Relay Solenoid Door Robot"
    ImageSwitcher (31,63 15x15), variable: InputOutput_GVL.xIn1401, behaviour: TOGGLE
    ImageSwitcher (31,85 15x15), variable: InputOutput_GVL.xIn1402, behaviour: TOGGLE
    ImageSwitcher (31,106 15x15), variable: InputOutput_GVL.xIn1403, behaviour: TOGGLE
    ImageSwitcher (31,127 15x15), variable: InputOutput_GVL.xIn1404, behaviour: TOGGLE
    ImageSwitcher (31,148 15x15), variable: InputOutput_GVL.xIn1405, behaviour: TOGGLE
    ImageSwitcher (31,170 15x15), variable: InputOutput_GVL.xIn1406, behaviour: TOGGLE
    ImageSwitcher (31,191 15x15), variable: InputOutput_GVL.xIn1407, behaviour: TOGGLE
    ImageSwitcher (31,214 15x15), variable: InputOutput_GVL.xIn1408, behaviour: TOGGLE
    ImageSwitcher (31,235 15x15), variable: InputOutput_GVL.xIn1409, behaviour: TOGGLE
    ImageSwitcher (31,257 15x15), variable: InputOutput_GVL.xIn1410, behaviour: TOGGLE
    ImageSwitcher (31,278 15x15), variable: InputOutput_GVL.xIn1411, behaviour: TOGGLE
    ImageSwitcher (31,299 15x15), variable: InputOutput_GVL.xIn1412, behaviour: TOGGLE
    ImageSwitcher (31,320 15x15), variable: InputOutput_GVL.xIn1413, behaviour: TOGGLE
    ImageSwitcher (31,342 15x15), variable: InputOutput_GVL.xIn1414, behaviour: TOGGLE
    ImageSwitcher (31,363 15x15), variable: InputOutput_GVL.xIn1415, behaviour: TOGGLE
    Button (769,-1 30x30), image: VisuSymbols.Symbols.Wrong
        OnMouseClick: CloseDialog Dialog=P1_DI3, Result=OK, NumpadKeypadSet=True
END_VISUALIZATION

// ---- VISUs/PLC Status/P1 - Panel Robot/P1_DI4.TcVIS
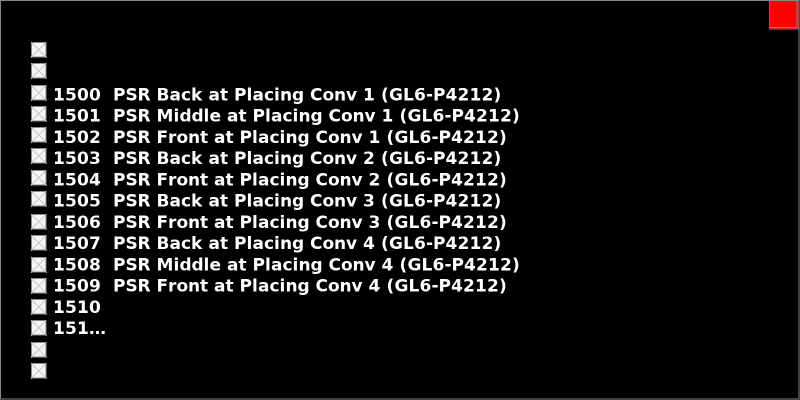
VISUALIZATION P1_DI4  // 800x400, background image 
    ImageSwitcher (31,42 15x15), variable: InputOutput_GVL.xIn1500, behaviour: TOGGLE
    Label (50,16 625x391), "1500 PSR Back at Placing Conv 1 (GL6-P4212) 1501 PSR Middle at Placing Conv 1 (GL6-P4212) 1502 PSR Front at Placing Conv 1 (GL6-P4212) 1503 PSR Back at Placing Conv 2 (GL6-P4212) 1504 PSR Front at Placing Conv 2 (GL6-P4212) 1505 PSR Back at Placing Conv 3 (GL6-P4212) 1506 PSR Front at Placing Conv 3 (GL6-P4212) 1507 PSR Back at Placing Conv 4 (GL6-P4212) 1508 PSR Middle at Placing Conv 4 (GL6-P4212) 1509 PSR Front at Placing Conv 4 (GL6-P4212) 1510 1511 1512 1513 1514 1515"
    ImageSwitcher (31,63 15x15), variable: InputOutput_GVL.xIn1501, behaviour: TOGGLE
    ImageSwitcher (31,85 15x15), variable: InputOutput_GVL.xIn1502, behaviour: TOGGLE
    ImageSwitcher (31,106 15x15), variable: InputOutput_GVL.xIn1503, behaviour: TOGGLE
    ImageSwitcher (31,127 15x15), variable: InputOutput_GVL.xIn1504, behaviour: TOGGLE
    ImageSwitcher (31,148 15x15), variable: InputOutput_GVL.xIn1505, behaviour: TOGGLE
    ImageSwitcher (31,170 15x15), variable: InputOutput_GVL.xIn1506, behaviour: TOGGLE
    ImageSwitcher (31,191 15x15), variable: InputOutput_GVL.xIn1507, behaviour: TOGGLE
    ImageSwitcher (31,214 15x15), variable: InputOutput_GVL.xIn1508, behaviour: TOGGLE
    ImageSwitcher (31,235 15x15), variable: InputOutput_GVL.xIn1509, behaviour: TOGGLE
    ImageSwitcher (31,257 15x15), variable: InputOutput_GVL.xIn1510, behaviour: TOGGLE
    ImageSwitcher (31,278 15x15), variable: InputOutput_GVL.xIn1511, behaviour: TOGGLE
    ImageSwitcher (31,299 15x15), variable: InputOutput_GVL.xIn1512, behaviour: TOGGLE
    ImageSwitcher (31,320 15x15), variable: InputOutput_GVL.xIn1513, behaviour: TOGGLE
    ImageSwitcher (31,342 15x15), variable: InputOutput_GVL.xIn1514, behaviour: TOGGLE
    ImageSwitcher (31,363 15x15), variable: InputOutput_GVL.xIn1515, behaviour: TOGGLE
    Button (769,-1 30x30), image: VisuSymbols.Symbols.Wrong
        OnMouseClick: CloseDialog Dialog=P1_DI4, Result=OK, NumpadKeypadSet=True
END_VISUALIZATION

// ---- VISUs/PLC Status/P1 - Panel Robot/P1_DO1.TcVIS
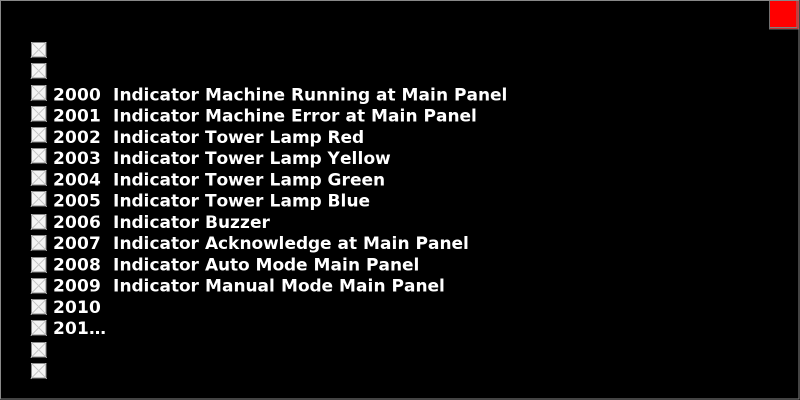
VISUALIZATION P1_DO1  // 800x400, background image 
    ImageSwitcher (31,42 15x15), variable: InputOutput_GVL.xIn1000, behaviour: TOGGLE
    Label (50,16 625x391), "2000 Indicator Machine Running at Main Panel 2001 Indicator Machine Error at Main Panel 2002 Indicator Tower Lamp Red 2003 Indicator Tower Lamp Yellow 2004 Indicator Tower Lamp Green 2005 Indicator Tower Lamp Blue 2006 Indicator Buzzer 2007 Indicator Acknowledge at Main Panel 2008 Indicator Auto Mode Main Panel 2009 Indicator Manual Mode Main Panel 2010 2011 2012 2013 2014 2015"
    ImageSwitcher (31,63 15x15), variable: InputOutput_GVL.xIn1001, behaviour: TOGGLE
    ImageSwitcher (31,85 15x15), variable: InputOutput_GVL.xIn1002, behaviour: TOGGLE
    ImageSwitcher (31,106 15x15), variable: InputOutput_GVL.xIn1003, behaviour: TOGGLE
    ImageSwitcher (31,127 15x15), variable: InputOutput_GVL.xIn1004, behaviour: TOGGLE
    ImageSwitcher (31,148 15x15), variable: InputOutput_GVL.xIn1005, behaviour: TOGGLE
    ImageSwitcher (31,170 15x15), variable: InputOutput_GVL.xIn1006, behaviour: TOGGLE
    ImageSwitcher (31,191 15x15), variable: InputOutput_GVL.xIn1007, behaviour: TOGGLE
    ImageSwitcher (31,214 15x15), variable: InputOutput_GVL.xIn1008, behaviour: TOGGLE
    ImageSwitcher (31,235 15x15), variable: InputOutput_GVL.xIn1009, behaviour: TOGGLE
    ImageSwitcher (31,257 15x15), variable: InputOutput_GVL.xIn1010, behaviour: TOGGLE
    ImageSwitcher (31,278 15x15), variable: InputOutput_GVL.xIn1011, behaviour: TOGGLE
    ImageSwitcher (31,299 15x15), variable: InputOutput_GVL.xIn1012, behaviour: TOGGLE
    ImageSwitcher (31,320 15x15), variable: InputOutput_GVL.xIn1013, behaviour: TOGGLE
    ImageSwitcher (31,342 15x15), variable: InputOutput_GVL.xIn1014, behaviour: TOGGLE
    ImageSwitcher (31,363 15x15), variable: InputOutput_GVL.xIn1015, behaviour: TOGGLE
    Button (769,-1 30x30), image: VisuSymbols.Symbols.Wrong
        OnMouseClick: CloseDialog Dialog=P1_DO1, Result=OK, NumpadKeypadSet=True
END_VISUALIZATION

// ---- VISUs/PLC Status/P1 - Panel Robot/P1_DO2.TcVIS
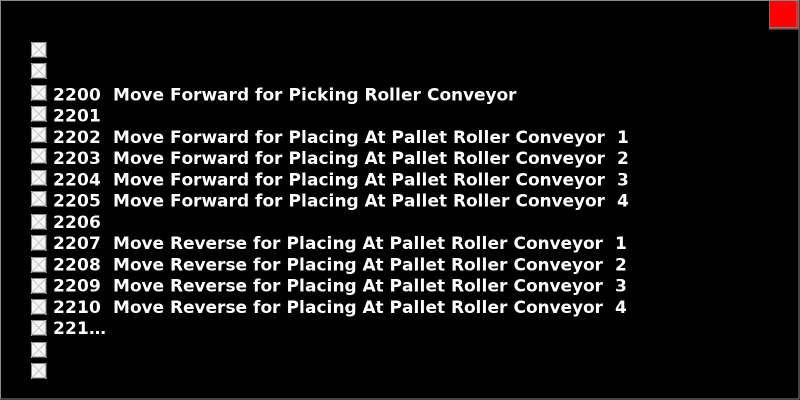
VISUALIZATION P1_DO2  // 800x400, background image 
    ImageSwitcher (31,42 15x15), variable: InputOutput_GVL.xIn1000, behaviour: TOGGLE
    Label (50,16 625x391), "2200 Move Forward for Picking Roller Conveyor 2201 2202 Move Forward for Placing At Pallet Roller Conveyor 1 2203 Move Forward for Placing At Pallet Roller Conveyor 2 2204 Move Forward for Placing At Pallet Roller Conveyor 3 2205 Move Forward for Placing At Pallet Roller Conveyor 4 2206 2207 Move Reverse for Placing At Pallet Roller Conveyor 1 2208 Move Reverse for Placing At Pallet Roller Conveyor 2 2209 Move Reverse for Placing At Pallet Roller Conveyor 3 2210 Move Reverse for Placing At Pallet Roller Conveyor 4 2211 2212 2213 2214 2215 Reset Error for All Inverter at P1, Relay"
    ImageSwitcher (31,63 15x15), variable: InputOutput_GVL.xIn1001, behaviour: TOGGLE
    ImageSwitcher (31,85 15x15), variable: InputOutput_GVL.xIn1002, behaviour: TOGGLE
    ImageSwitcher (31,106 15x15), variable: InputOutput_GVL.xIn1003, behaviour: TOGGLE
    ImageSwitcher (31,127 15x15), variable: InputOutput_GVL.xIn1004, behaviour: TOGGLE
    ImageSwitcher (31,148 15x15), variable: InputOutput_GVL.xIn1005, behaviour: TOGGLE
    ImageSwitcher (31,170 15x15), variable: InputOutput_GVL.xIn1006, behaviour: TOGGLE
    ImageSwitcher (31,191 15x15), variable: InputOutput_GVL.xIn1007, behaviour: TOGGLE
    ImageSwitcher (31,214 15x15), variable: InputOutput_GVL.xIn1008, behaviour: TOGGLE
    ImageSwitcher (31,235 15x15), variable: InputOutput_GVL.xIn1009, behaviour: TOGGLE
    ImageSwitcher (31,257 15x15), variable: InputOutput_GVL.xIn1010, behaviour: TOGGLE
    ImageSwitcher (31,278 15x15), variable: InputOutput_GVL.xIn1011, behaviour: TOGGLE
    ImageSwitcher (31,299 15x15), variable: InputOutput_GVL.xIn1012, behaviour: TOGGLE
    ImageSwitcher (31,320 15x15), variable: InputOutput_GVL.xIn1013, behaviour: TOGGLE
    ImageSwitcher (31,342 15x15), variable: InputOutput_GVL.xIn1014, behaviour: TOGGLE
    ImageSwitcher (31,363 15x15), variable: InputOutput_GVL.xIn1015, behaviour: TOGGLE
    Button (769,-1 30x30), image: VisuSymbols.Symbols.Wrong
        OnMouseClick: CloseDialog Dialog=P1_DO2, Result=OK, NumpadKeypadSet=True
END_VISUALIZATION

// ---- VISUs/PLC Status/P1 - Panel Robot/P1_DO3.TcVIS
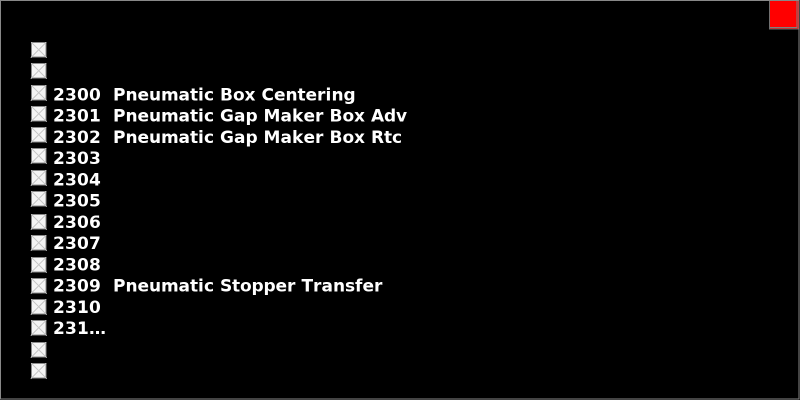
VISUALIZATION P1_DO3  // 800x400, background image 
    ImageSwitcher (31,42 15x15), variable: InputOutput_GVL.xIn1000, behaviour: TOGGLE
    Label (50,16 625x391), "2300 Pneumatic Box Centering 2301 Pneumatic Gap Maker Box Adv 2302 Pneumatic Gap Maker Box Rtc 2303 2304 2305 2306 2307 2308 2309 Pneumatic Stopper Transfer 2310 2311 2312 2313 2314 Status Solenoid Door Robot 2315 Release Solenoid Door Robot"
    ImageSwitcher (31,63 15x15), variable: InputOutput_GVL.xIn1001, behaviour: TOGGLE
    ImageSwitcher (31,85 15x15), variable: InputOutput_GVL.xIn1002, behaviour: TOGGLE
    ImageSwitcher (31,106 15x15), variable: InputOutput_GVL.xIn1003, behaviour: TOGGLE
    ImageSwitcher (31,127 15x15), variable: InputOutput_GVL.xIn1004, behaviour: TOGGLE
    ImageSwitcher (31,148 15x15), variable: InputOutput_GVL.xIn1005, behaviour: TOGGLE
    ImageSwitcher (31,170 15x15), variable: InputOutput_GVL.xIn1006, behaviour: TOGGLE
    ImageSwitcher (31,191 15x15), variable: InputOutput_GVL.xIn1007, behaviour: TOGGLE
    ImageSwitcher (31,214 15x15), variable: InputOutput_GVL.xIn1008, behaviour: TOGGLE
    ImageSwitcher (31,235 15x15), variable: InputOutput_GVL.xIn1009, behaviour: TOGGLE
    ImageSwitcher (31,257 15x15), variable: InputOutput_GVL.xIn1010, behaviour: TOGGLE
    ImageSwitcher (31,278 15x15), variable: InputOutput_GVL.xIn1011, behaviour: TOGGLE
    ImageSwitcher (31,299 15x15), variable: InputOutput_GVL.xIn1012, behaviour: TOGGLE
    ImageSwitcher (31,320 15x15), variable: InputOutput_GVL.xIn1013, behaviour: TOGGLE
    ImageSwitcher (31,342 15x15), variable: InputOutput_GVL.xIn1014, behaviour: TOGGLE
    ImageSwitcher (31,363 15x15), variable: InputOutput_GVL.xIn1015, behaviour: TOGGLE
    Button (769,-1 30x30), image: VisuSymbols.Symbols.Wrong
        OnMouseClick: CloseDialog Dialog=P1_DO3, Result=OK, NumpadKeypadSet=True
END_VISUALIZATION

// ---- VISUs/PLC Status/P2 - Panel Outfeed/P2_DI1.TcVIS
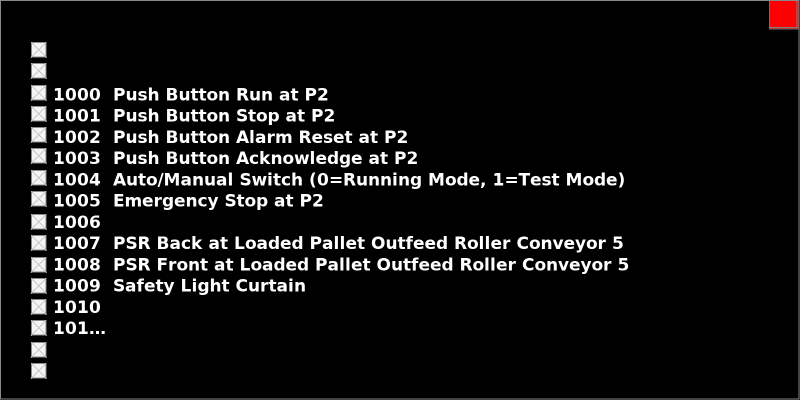
VISUALIZATION P2_DI1  // 800x400, background image 
    ImageSwitcher (31,42 15x15), variable: InputOutput_GVL.Digital_Input[1], behaviour: TOGGLE
    Label (50,16 724x391), "1000 Push Button Run at P2 1001 Push Button Stop at P2 1002 Push Button Alarm Reset at P2 1003 Push Button Acknowledge at P2 1004 Auto/Manual Switch (0=Running Mode, 1=Test Mode) 1005 Emergency Stop at P2 1006 1007 PSR Back at Loaded Pallet Outfeed Roller Conveyor 5 1008 PSR Front at Loaded Pallet Outfeed Roller Conveyor 5 1009 Safety Light Curtain 1010 1011 1012 1013 PSR Back at Detect Loaded Pallet Buffer Roller Conv 2 1014 PSR Front at Detect Loaded Pallet Buffer Roller Conv 2 1015 Feedback Loaded Pallet Outfeed Roller Conveyor 5 is Running"
    ImageSwitcher (31,63 15x15), variable: InputOutput_GVL.Digital_Input[2], behaviour: TOGGLE
    ImageSwitcher (31,85 15x15), variable: InputOutput_GVL.Digital_Input[3], behaviour: TOGGLE
    ImageSwitcher (31,106 15x15), variable: InputOutput_GVL.Digital_Input[4], behaviour: TOGGLE
    ImageSwitcher (31,127 15x15), variable: InputOutput_GVL.Digital_Input[5], behaviour: TOGGLE
    ImageSwitcher (31,148 15x15), variable: InputOutput_GVL.Digital_Input[6], behaviour: TOGGLE
    ImageSwitcher (31,170 15x15), variable: InputOutput_GVL.Digital_Input[7], behaviour: TOGGLE
    ImageSwitcher (31,191 15x15), variable: InputOutput_GVL.Digital_Input[8], behaviour: TOGGLE
    ImageSwitcher (31,214 15x15), variable: InputOutput_GVL.Digital_Input[9], behaviour: TOGGLE
    ImageSwitcher (31,235 15x15), variable: InputOutput_GVL.Digital_Input[10], behaviour: TOGGLE
    ImageSwitcher (31,257 15x15), variable: InputOutput_GVL.Digital_Input[11], behaviour: TOGGLE
    ImageSwitcher (31,278 15x15), variable: InputOutput_GVL.Digital_Input[12], behaviour: TOGGLE
    ImageSwitcher (31,299 15x15), variable: InputOutput_GVL.Digital_Input[13], behaviour: TOGGLE
    ImageSwitcher (31,320 15x15), variable: InputOutput_GVL.Digital_Input[14], behaviour: TOGGLE
    ImageSwitcher (31,342 15x15), variable: InputOutput_GVL.Digital_Input[15], behaviour: TOGGLE
    ImageSwitcher (31,363 15x15), variable: InputOutput_GVL.Digital_Input[16], behaviour: TOGGLE
    Button (769,-1 30x30), image: VisuSymbols.Symbols.Wrong
        OnMouseClick: CloseDialog Dialog=P2_DI1, Result=OK, NumpadKeypadSet=True
END_VISUALIZATION

// ---- VISUs/PLC Status/P2 - Panel Outfeed/P2_DI2.TcVIS
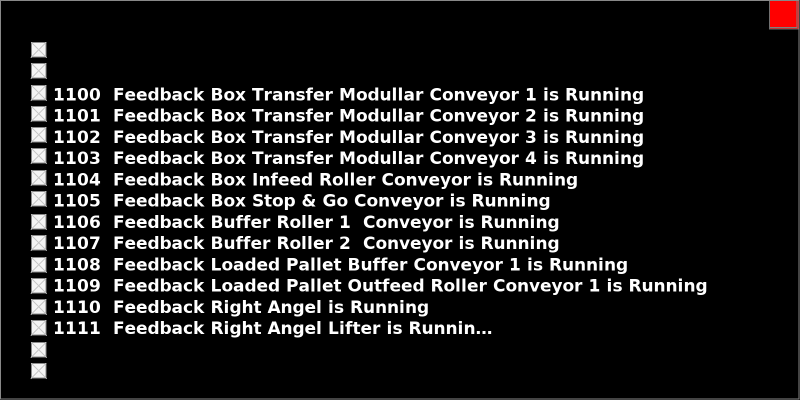
VISUALIZATION P2_DI2  // 800x400, background image 
    ImageSwitcher (31,42 15x15), variable: InputOutput_GVL.Digital_Input[17], behaviour: TOGGLE
    Label (50,16 720x391), "1100 Feedback Box Transfer Modullar Conveyor 1 is Running 1101 Feedback Box Transfer Modullar Conveyor 2 is Running 1102 Feedback Box Transfer Modullar Conveyor 3 is Running 1103 Feedback Box Transfer Modullar Conveyor 4 is Running 1104 Feedback Box Infeed Roller Conveyor is Running 1105 Feedback Box Stop & Go Conveyor is Running 1106 Feedback Buffer Roller 1 Conveyor is Running 1107 Feedback Buffer Roller 2 Conveyor is Running 1108 Feedback Loaded Pallet Buffer Conveyor 1 is Running 1109 Feedback Loaded Pallet Outfeed Roller Conveyor 1 is Running 1110 Feedback Right Angel is Running 1111 Feedback Right Angel Lifter is Running 1112 Feedback Loaded Pallet Outfeed Roller Conveyor 2 is Running 1113 Feedback Loaded Pallet Outfeed Roller Conveyor 3 is Running 1114 Feedback Loaded Pallet Outfeed Roller Conveyor 4 is Running 1115 Feedback Loaded Pallet Buffer 2 is Running"
    ImageSwitcher (31,63 15x15), variable: InputOutput_GVL.Digital_Input[18], behaviour: TOGGLE
    ImageSwitcher (31,85 15x15), variable: InputOutput_GVL.Digital_Input[19], behaviour: TOGGLE
    ImageSwitcher (31,106 15x15), variable: InputOutput_GVL.Digital_Input[20], behaviour: TOGGLE
    ImageSwitcher (31,127 15x15), variable: InputOutput_GVL.Digital_Input[21], behaviour: TOGGLE
    ImageSwitcher (31,148 15x15), variable: InputOutput_GVL.Digital_Input[22], behaviour: TOGGLE
    ImageSwitcher (31,170 15x15), variable: InputOutput_GVL.Digital_Input[23], behaviour: TOGGLE
    ImageSwitcher (31,191 15x15), variable: InputOutput_GVL.Digital_Input[24], behaviour: TOGGLE
    ImageSwitcher (31,214 15x15), variable: InputOutput_GVL.Digital_Input[25], behaviour: TOGGLE
    ImageSwitcher (31,235 15x15), variable: InputOutput_GVL.Digital_Input[26], behaviour: TOGGLE
    ImageSwitcher (31,257 15x15), variable: InputOutput_GVL.Digital_Input[27], behaviour: TOGGLE
    ImageSwitcher (31,278 15x15), variable: InputOutput_GVL.Digital_Input[28], behaviour: TOGGLE
    ImageSwitcher (31,299 15x15), variable: InputOutput_GVL.Digital_Input[29], behaviour: TOGGLE
    ImageSwitcher (31,320 15x15), variable: InputOutput_GVL.Digital_Input[30], behaviour: TOGGLE
    ImageSwitcher (31,342 15x15), variable: InputOutput_GVL.Digital_Input[31], behaviour: TOGGLE
    ImageSwitcher (31,363 15x15), variable: InputOutput_GVL.Digital_Input[32], behaviour: TOGGLE
    Button (769,-1 30x30), image: VisuSymbols.Symbols.Wrong
        OnMouseClick: CloseDialog Dialog=P2_DI2, Result=OK, NumpadKeypadSet=True
END_VISUALIZATION

// ---- VISUs/PLC Status/P2 - Panel Outfeed/P2_DI3.TcVIS
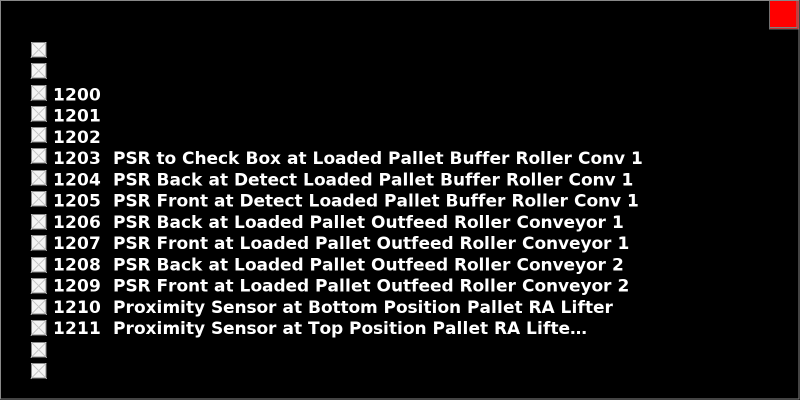
VISUALIZATION P2_DI3  // 800x400, background image 
    ImageSwitcher (31,42 15x15), variable: InputOutput_GVL.Digital_Input[33], behaviour: TOGGLE
    Label (50,16 687x391), "1200 1201 1202 1203 PSR to Check Box at Loaded Pallet Buffer Roller Conv 1 1204 PSR Back at Detect Loaded Pallet Buffer Roller Conv 1 1205 PSR Front at Detect Loaded Pallet Buffer Roller Conv 1 1206 PSR Back at Loaded Pallet Outfeed Roller Conveyor 1 1207 PSR Front at Loaded Pallet Outfeed Roller Conveyor 1 1208 PSR Back at Loaded Pallet Outfeed Roller Conveyor 2 1209 PSR Front at Loaded Pallet Outfeed Roller Conveyor 2 1210 Proximity Sensor at Bottom Position Pallet RA Lifter 1211 Proximity Sensor at Top Position Pallet RA Lifter 1212 PSR Back at Loaded Pallet Outfeed Roller Conveyor 3 1213 PSR Front at Loaded Pallet Outfeed Roller Conveyor 3 1214 PSR Back at Loaded Pallet Outfeed Roller Conveyor 4 1215 PSR Front at Loaded Pallet Outfeed Roller Conveyor 4"
    ImageSwitcher (31,63 15x15), variable: InputOutput_GVL.Digital_Input[34], behaviour: TOGGLE
    ImageSwitcher (31,85 15x15), variable: InputOutput_GVL.Digital_Input[35], behaviour: TOGGLE
    ImageSwitcher (31,106 15x15), variable: InputOutput_GVL.Digital_Input[36], behaviour: TOGGLE
    ImageSwitcher (31,127 15x15), variable: InputOutput_GVL.Digital_Input[37], behaviour: TOGGLE
    ImageSwitcher (31,148 15x15), variable: InputOutput_GVL.Digital_Input[38], behaviour: TOGGLE
    ImageSwitcher (31,170 15x15), variable: InputOutput_GVL.Digital_Input[39], behaviour: TOGGLE
    ImageSwitcher (31,191 15x15), variable: InputOutput_GVL.Digital_Input[40], behaviour: TOGGLE
    ImageSwitcher (31,214 15x15), variable: InputOutput_GVL.Digital_Input[41], behaviour: TOGGLE
    ImageSwitcher (31,235 15x15), variable: InputOutput_GVL.Digital_Input[42], behaviour: TOGGLE
    ImageSwitcher (31,257 15x15), variable: InputOutput_GVL.Digital_Input[43], behaviour: TOGGLE
    ImageSwitcher (31,278 15x15), variable: InputOutput_GVL.Digital_Input[44], behaviour: TOGGLE
    ImageSwitcher (31,299 15x15), variable: InputOutput_GVL.Digital_Input[45], behaviour: TOGGLE
    ImageSwitcher (31,320 15x15), variable: InputOutput_GVL.Digital_Input[46], behaviour: TOGGLE
    ImageSwitcher (31,342 15x15), variable: InputOutput_GVL.Digital_Input[47], behaviour: TOGGLE
    ImageSwitcher (31,363 15x15), variable: InputOutput_GVL.Digital_Input[48], behaviour: TOGGLE
    Button (769,-1 30x30), image: VisuSymbols.Symbols.Wrong
        OnMouseClick: CloseDialog Dialog=P2_DI3, Result=OK, NumpadKeypadSet=True
END_VISUALIZATION

// ---- VISUs/PLC Status/P2 - Panel Outfeed/P2_DI4.TcVIS
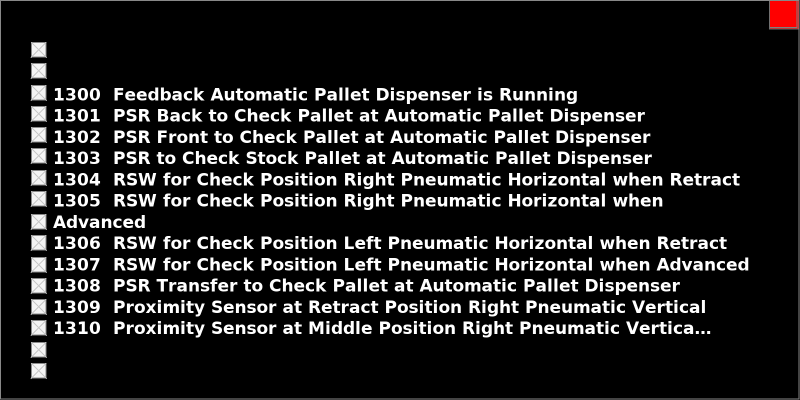
VISUALIZATION P2_DI4  // 800x400, background image 
    ImageSwitcher (31,42 15x15), variable: InputOutput_GVL.Digital_Input[49], behaviour: TOGGLE
    Label (50,16 705x391), "1300 Feedback Automatic Pallet Dispenser is Running 1301 PSR Back to Check Pallet at Automatic Pallet Dispenser 1302 PSR Front to Check Pallet at Automatic Pallet Dispenser 1303 PSR to Check Stock Pallet at Automatic Pallet Dispenser 1304 RSW for Check Position Right Pneumatic Horizontal when Retract 1305 RSW for Check Position Right Pneumatic Horizontal when Advanced 1306 RSW for Check Position Left Pneumatic Horizontal when Retract 1307 RSW for Check Position Left Pneumatic Horizontal when Advanced 1308 PSR Transfer to Check Pallet at Automatic Pallet Dispenser 1309 Proximity Sensor at Retract Position Right Pneumatic Vertical 1310 Proximity Sensor at Middle Position Right Pneumatic Vertical 1311 Proximity Sensor at Advanced Position Right Pneumatic Vertical 1312 Proximity Sensor at Retract Position Left Pneumatic Vertical 1313 Proximity Sensor at Middle Position Left Pneumatic Vertical 1314 Proximity Sensor at Advanced Position Left Pneumatic Vertical 1315 Request Release Solenoid Door Outfeed"
    ImageSwitcher (31,63 15x15), variable: InputOutput_GVL.Digital_Input[50], behaviour: TOGGLE
    ImageSwitcher (31,85 15x15), variable: InputOutput_GVL.Digital_Input[51], behaviour: TOGGLE
    ImageSwitcher (31,106 15x15), variable: InputOutput_GVL.Digital_Input[52], behaviour: TOGGLE
    ImageSwitcher (31,127 15x15), variable: InputOutput_GVL.Digital_Input[53], behaviour: TOGGLE
    ImageSwitcher (31,148 15x15), variable: InputOutput_GVL.Digital_Input[54], behaviour: TOGGLE
    ImageSwitcher (31,170 15x15), variable: InputOutput_GVL.Digital_Input[55], behaviour: TOGGLE
    ImageSwitcher (31,191 15x15), variable: InputOutput_GVL.Digital_Input[56], behaviour: TOGGLE
    ImageSwitcher (31,214 15x15), variable: InputOutput_GVL.Digital_Input[57], behaviour: TOGGLE
    ImageSwitcher (31,235 15x15), variable: InputOutput_GVL.Digital_Input[58], behaviour: TOGGLE
    ImageSwitcher (31,257 15x15), variable: InputOutput_GVL.Digital_Input[59], behaviour: TOGGLE
    ImageSwitcher (31,278 15x15), variable: InputOutput_GVL.Digital_Input[60], behaviour: TOGGLE
    ImageSwitcher (31,299 15x15), variable: InputOutput_GVL.Digital_Input[61], behaviour: TOGGLE
    ImageSwitcher (31,320 15x15), variable: InputOutput_GVL.Digital_Input[62], behaviour: TOGGLE
    ImageSwitcher (31,342 15x15), variable: InputOutput_GVL.Digital_Input[63], behaviour: TOGGLE
    ImageSwitcher (31,363 15x15), variable: InputOutput_GVL.Digital_Input[64], behaviour: TOGGLE
    Button (769,-1 30x30), image: VisuSymbols.Symbols.Wrong
        OnMouseClick: CloseDialog Dialog=P2_DI4, Result=OK, NumpadKeypadSet=True
END_VISUALIZATION

// ---- VISUs/PLC Status/P2 - Panel Outfeed/P2_DI5.TcVIS
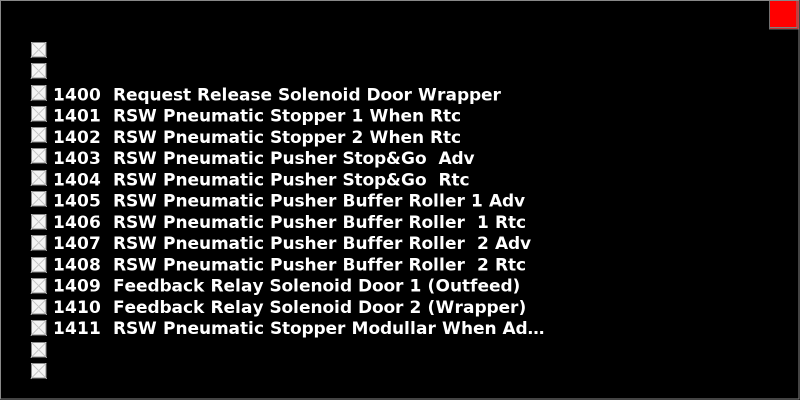
VISUALIZATION P2_DI5  // 800x400, background image 
    ImageSwitcher (31,42 15x15), variable: InputOutput_GVL.Digital_Input[65], behaviour: TOGGLE
    Label (50,16 625x391), "1400 Request Release Solenoid Door Wrapper 1401 RSW Pneumatic Stopper 1 When Rtc 1402 RSW Pneumatic Stopper 2 When Rtc 1403 RSW Pneumatic Pusher Stop&Go Adv 1404 RSW Pneumatic Pusher Stop&Go Rtc 1405 RSW Pneumatic Pusher Buffer Roller 1 Adv 1406 RSW Pneumatic Pusher Buffer Roller 1 Rtc 1407 RSW Pneumatic Pusher Buffer Roller 2 Adv 1408 RSW Pneumatic Pusher Buffer Roller 2 Rtc 1409 Feedback Relay Solenoid Door 1 (Outfeed) 1410 Feedback Relay Solenoid Door 2 (Wrapper) 1411 RSW Pneumatic Stopper Modullar When Adv 1412 RSW Pneumatic Stopper Modullar When Rtc 1413 1414 Interlock Feedback Pallet Ready at Infeed Dispenser 1415 Interlock Feedback Pallet Ready at Unloading"
    ImageSwitcher (31,63 15x15), variable: InputOutput_GVL.Digital_Input[66], behaviour: TOGGLE
    ImageSwitcher (31,85 15x15), variable: InputOutput_GVL.Digital_Input[67], behaviour: TOGGLE
    ImageSwitcher (31,106 15x15), variable: InputOutput_GVL.Digital_Input[68], behaviour: TOGGLE
    ImageSwitcher (31,127 15x15), variable: InputOutput_GVL.Digital_Input[69], behaviour: TOGGLE
    ImageSwitcher (31,148 15x15), variable: InputOutput_GVL.Digital_Input[70], behaviour: TOGGLE
    ImageSwitcher (31,170 15x15), variable: InputOutput_GVL.Digital_Input[71], behaviour: TOGGLE
    ImageSwitcher (31,191 15x15), variable: InputOutput_GVL.Digital_Input[72], behaviour: TOGGLE
    ImageSwitcher (31,214 15x15), variable: InputOutput_GVL.Digital_Input[73], behaviour: TOGGLE
    ImageSwitcher (31,235 15x15), variable: InputOutput_GVL.Digital_Input[74], behaviour: TOGGLE
    ImageSwitcher (31,257 15x15), variable: InputOutput_GVL.Digital_Input[75], behaviour: TOGGLE
    ImageSwitcher (31,278 15x15), variable: InputOutput_GVL.Digital_Input[76], behaviour: TOGGLE
    ImageSwitcher (31,299 15x15), variable: InputOutput_GVL.Digital_Input[77], behaviour: TOGGLE
    ImageSwitcher (31,320 15x15), variable: InputOutput_GVL.Digital_Input[78], behaviour: TOGGLE
    ImageSwitcher (31,342 15x15), variable: InputOutput_GVL.Digital_Input[79], behaviour: TOGGLE
    ImageSwitcher (31,363 15x15), variable: InputOutput_GVL.Digital_Input[80], behaviour: TOGGLE
    Button (769,-1 30x30), image: VisuSymbols.Symbols.Wrong
        OnMouseClick: CloseDialog Dialog=P2_DI5, Result=OK, NumpadKeypadSet=True
END_VISUALIZATION

// ---- VISUs/PLC Status/P2 - Panel Outfeed/P2_DI6.TcVIS
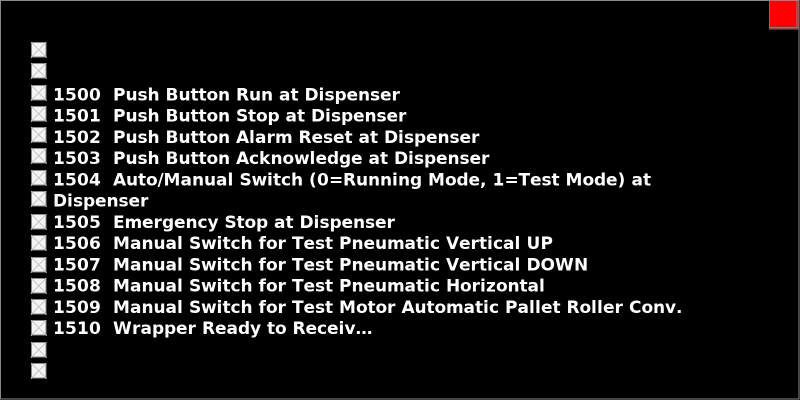
VISUALIZATION P2_DI6  // 800x400, background image 
    ImageSwitcher (31,42 15x15), variable: InputOutput_GVL.Digital_Input[81], behaviour: TOGGLE
    Label (50,16 677x391), "1500 Push Button Run at Dispenser 1501 Push Button Stop at Dispenser 1502 Push Button Alarm Reset at Dispenser 1503 Push Button Acknowledge at Dispenser 1504 Auto/Manual Switch (0=Running Mode, 1=Test Mode) at Dispenser 1505 Emergency Stop at Dispenser 1506 Manual Switch for Test Pneumatic Vertical UP 1507 Manual Switch for Test Pneumatic Vertical DOWN 1508 Manual Switch for Test Pneumatic Horizontal 1509 Manual Switch for Test Motor Automatic Pallet Roller Conv. 1510 Wrapper Ready to Receive 1511 End of Transfer Pallet in Infeed 1512 Pallet Ready in Outfeed 1513 Emergency Stop Wrapper is Active 1514 Status Bypass Wrapper Existing 1515 Pressure Switch for Pallet Dispenser"
    ImageSwitcher (31,63 15x15), variable: InputOutput_GVL.Digital_Input[82], behaviour: TOGGLE
    ImageSwitcher (31,85 15x15), variable: InputOutput_GVL.Digital_Input[83], behaviour: TOGGLE
    ImageSwitcher (31,106 15x15), variable: InputOutput_GVL.Digital_Input[84], behaviour: TOGGLE
    ImageSwitcher (31,127 15x15), variable: InputOutput_GVL.Digital_Input[85], behaviour: TOGGLE
    ImageSwitcher (31,148 15x15), variable: InputOutput_GVL.Digital_Input[86], behaviour: TOGGLE
    ImageSwitcher (31,170 15x15), variable: InputOutput_GVL.Digital_Input[87], behaviour: TOGGLE
    ImageSwitcher (31,191 15x15), variable: InputOutput_GVL.Digital_Input[88], behaviour: TOGGLE
    ImageSwitcher (31,214 15x15), variable: InputOutput_GVL.Digital_Input[89], behaviour: TOGGLE
    ImageSwitcher (31,235 15x15), variable: InputOutput_GVL.Digital_Input[90], behaviour: TOGGLE
    ImageSwitcher (31,257 15x15), variable: InputOutput_GVL.Digital_Input[91], behaviour: TOGGLE
    ImageSwitcher (31,278 15x15), variable: InputOutput_GVL.Digital_Input[92], behaviour: TOGGLE
    ImageSwitcher (31,299 15x15), variable: InputOutput_GVL.Digital_Input[93], behaviour: TOGGLE
    ImageSwitcher (31,320 15x15), variable: InputOutput_GVL.Digital_Input[94], behaviour: TOGGLE
    ImageSwitcher (31,342 15x15), variable: InputOutput_GVL.Digital_Input[95], behaviour: TOGGLE
    ImageSwitcher (31,363 15x15), variable: InputOutput_GVL.Digital_Input[96], behaviour: TOGGLE
    Button (769,-1 30x30), image: VisuSymbols.Symbols.Wrong
        OnMouseClick: CloseDialog Dialog=P2_DI6, Result=OK, NumpadKeypadSet=True
END_VISUALIZATION

// ---- VISUs/PLC Status/P2 - Panel Outfeed/P2_DI7.TcVIS
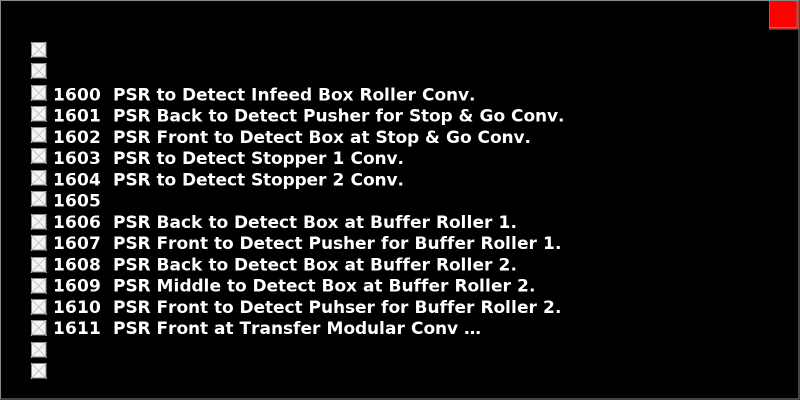
VISUALIZATION P2_DI7  // 800x400, background image 
    ImageSwitcher (31,42 15x15), variable: InputOutput_GVL.Digital_Input[97], behaviour: TOGGLE
    Label (50,16 696x391), "1600 PSR to Detect Infeed Box Roller Conv. 1601 PSR Back to Detect Pusher for Stop & Go Conv. 1602 PSR Front to Detect Box at Stop & Go Conv. 1603 PSR to Detect Stopper 1 Conv. 1604 PSR to Detect Stopper 2 Conv. 1605 1606 PSR Back to Detect Box at Buffer Roller 1. 1607 PSR Front to Detect Pusher for Buffer Roller 1. 1608 PSR Back to Detect Box at Buffer Roller 2. 1609 PSR Middle to Detect Box at Buffer Roller 2. 1610 PSR Front to Detect Puhser for Buffer Roller 2. 1611 PSR Front at Transfer Modular Conv 4 1612 PSR Front at Transfer Modular Conv 2 1613 PSR Back at Transfer Modular Conv 3 1614 PSR Front at Transfer Modular Conv 3 1615 PSR Back at Transfer Modular Conv 4"
    ImageSwitcher (31,63 15x15), variable: InputOutput_GVL.Digital_Input[98], behaviour: TOGGLE
    ImageSwitcher (31,85 15x15), variable: InputOutput_GVL.Digital_Input[99], behaviour: TOGGLE
    ImageSwitcher (31,106 15x15), variable: InputOutput_GVL.Digital_Input[100], behaviour: TOGGLE
    ImageSwitcher (31,127 15x15), variable: InputOutput_GVL.Digital_Input[101], behaviour: TOGGLE
    ImageSwitcher (31,148 15x15), variable: InputOutput_GVL.Digital_Input[102], behaviour: TOGGLE
    ImageSwitcher (31,170 15x15), variable: InputOutput_GVL.Digital_Input[103], behaviour: TOGGLE
    ImageSwitcher (31,191 15x15), variable: InputOutput_GVL.Digital_Input[104], behaviour: TOGGLE
    ImageSwitcher (31,214 15x15), variable: InputOutput_GVL.Digital_Input[105], behaviour: TOGGLE
    ImageSwitcher (31,235 15x15), variable: InputOutput_GVL.Digital_Input[106], behaviour: TOGGLE
    ImageSwitcher (31,257 15x15), variable: InputOutput_GVL.Digital_Input[107], behaviour: TOGGLE
    ImageSwitcher (31,278 15x15), variable: InputOutput_GVL.Digital_Input[108], behaviour: TOGGLE
    ImageSwitcher (31,299 15x15), variable: InputOutput_GVL.Digital_Input[109], behaviour: TOGGLE
    ImageSwitcher (31,320 15x15), variable: InputOutput_GVL.Digital_Input[110], behaviour: TOGGLE
    ImageSwitcher (31,342 15x15), variable: InputOutput_GVL.Digital_Input[111], behaviour: TOGGLE
    ImageSwitcher (31,363 15x15), variable: InputOutput_GVL.Digital_Input[112], behaviour: TOGGLE
    Button (769,-1 30x30), image: VisuSymbols.Symbols.Wrong
        OnMouseClick: CloseDialog Dialog=P2_DI7, Result=OK, NumpadKeypadSet=True
END_VISUALIZATION

// ---- VISUs/PLC Status/P2 - Panel Outfeed/P2_DO1.TcVIS
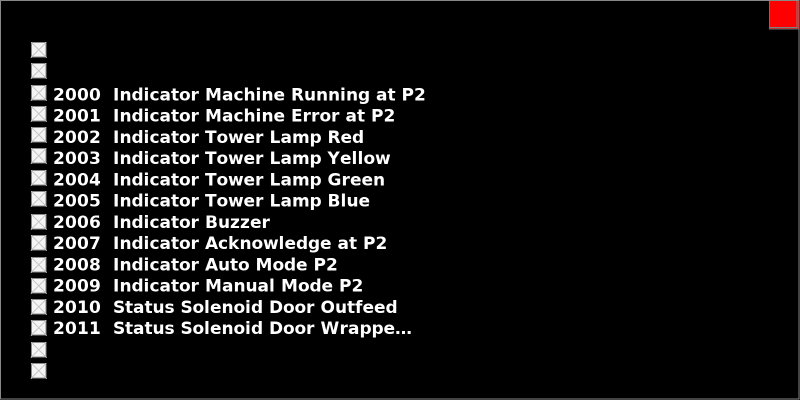
VISUALIZATION P2_DO1  // 800x400, background image 
    ImageSwitcher (31,42 15x15), variable: InputOutput_GVL.Digital_Output[1], behaviour: TOGGLE
    Label (50,16 625x391), "2000 Indicator Machine Running at P2 2001 Indicator Machine Error at P2 2002 Indicator Tower Lamp Red 2003 Indicator Tower Lamp Yellow 2004 Indicator Tower Lamp Green 2005 Indicator Tower Lamp Blue 2006 Indicator Buzzer 2007 Indicator Acknowledge at P2 2008 Indicator Auto Mode P2 2009 Indicator Manual Mode P2 2010 Status Solenoid Door Outfeed 2011 Status Solenoid Door Wrapper 2012 2013 Pneumatic Stopper Modullar Adv 2014 Pneumatic Stopper Modullar Rtc 2015 Move Forward for Loaded Pallet Outfeed Roller Conveyor 5"
    ImageSwitcher (31,63 15x15), variable: InputOutput_GVL.Digital_Output[2], behaviour: TOGGLE
    ImageSwitcher (31,85 15x15), variable: InputOutput_GVL.Digital_Output[3], behaviour: TOGGLE
    ImageSwitcher (31,106 15x15), variable: InputOutput_GVL.Digital_Output[4], behaviour: TOGGLE
    ImageSwitcher (31,127 15x15), variable: InputOutput_GVL.Digital_Output[5], behaviour: TOGGLE
    ImageSwitcher (31,148 15x15), variable: InputOutput_GVL.Digital_Output[6], behaviour: TOGGLE
    ImageSwitcher (31,170 15x15), variable: InputOutput_GVL.Digital_Output[7], behaviour: TOGGLE
    ImageSwitcher (31,191 15x15), variable: InputOutput_GVL.Digital_Output[8], behaviour: TOGGLE
    ImageSwitcher (31,214 15x15), variable: InputOutput_GVL.Digital_Output[9], behaviour: TOGGLE
    ImageSwitcher (31,235 15x15), variable: InputOutput_GVL.Digital_Output[10], behaviour: TOGGLE
    ImageSwitcher (31,257 15x15), variable: InputOutput_GVL.Digital_Output[11], behaviour: TOGGLE
    ImageSwitcher (31,278 15x15), variable: InputOutput_GVL.Digital_Output[12], behaviour: TOGGLE
    ImageSwitcher (31,299 15x15), variable: InputOutput_GVL.Digital_Output[13], behaviour: TOGGLE
    ImageSwitcher (31,320 15x15), variable: InputOutput_GVL.Digital_Output[14], behaviour: TOGGLE
    ImageSwitcher (31,342 15x15), variable: InputOutput_GVL.Digital_Output[15], behaviour: TOGGLE
    ImageSwitcher (31,363 15x15), variable: InputOutput_GVL.Digital_Output[16], behaviour: TOGGLE
    Button (769,-1 30x30), image: VisuSymbols.Symbols.Wrong
        OnMouseClick: CloseDialog Dialog=P2_DO1, Result=OK, NumpadKeypadSet=True
END_VISUALIZATION

// ---- VISUs/PLC Status/P2 - Panel Outfeed/P2_DO2.TcVIS
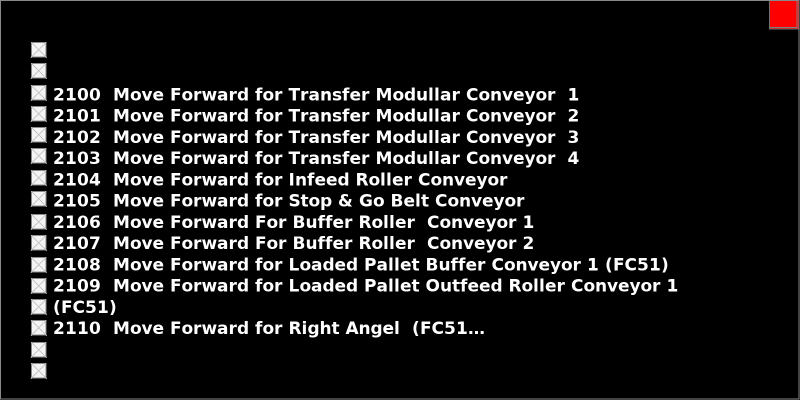
VISUALIZATION P2_DO2  // 800x400, background image 
    ImageSwitcher (31,42 15x15), variable: InputOutput_GVL.Digital_Output[17], behaviour: TOGGLE
    Label (50,16 668x391), "2100 Move Forward for Transfer Modullar Conveyor 1 2101 Move Forward for Transfer Modullar Conveyor 2 2102 Move Forward for Transfer Modullar Conveyor 3 2103 Move Forward for Transfer Modullar Conveyor 4 2104 Move Forward for Infeed Roller Conveyor 2105 Move Forward for Stop & Go Belt Conveyor 2106 Move Forward For Buffer Roller Conveyor 1 2107 Move Forward For Buffer Roller Conveyor 2 2108 Move Forward for Loaded Pallet Buffer Conveyor 1 (FC51) 2109 Move Forward for Loaded Pallet Outfeed Roller Conveyor 1 (FC51) 2110 Move Forward for Right Angel (FC51) 2111 Move Forward for Right Angel Lifter (FC51) 2112 Move Forward for Loaded Pallet Outfeed Roller Conveyor (FC51) 2113 Move Forward for Loaded Pallet Outfeed Roller Conveyor (FC51) 2114 Move Forward for Loaded Pallet Outfeed Roller Conveyor (FC51) 2115 Reset Error for All Inverter at P2, Relay"
    ImageSwitcher (31,63 15x15), variable: InputOutput_GVL.Digital_Output[18], behaviour: TOGGLE
    ImageSwitcher (31,85 15x15), variable: InputOutput_GVL.Digital_Output[19], behaviour: TOGGLE
    ImageSwitcher (31,106 15x15), variable: InputOutput_GVL.Digital_Output[20], behaviour: TOGGLE
    ImageSwitcher (31,127 15x15), variable: InputOutput_GVL.Digital_Output[21], behaviour: TOGGLE
    ImageSwitcher (31,148 15x15), variable: InputOutput_GVL.Digital_Output[22], behaviour: TOGGLE
    ImageSwitcher (31,170 15x15), variable: InputOutput_GVL.Digital_Output[23], behaviour: TOGGLE
    ImageSwitcher (31,191 15x15), variable: InputOutput_GVL.Digital_Output[24], behaviour: TOGGLE
    ImageSwitcher (31,214 15x15), variable: InputOutput_GVL.Digital_Output[25], behaviour: TOGGLE
    ImageSwitcher (31,235 15x15), variable: InputOutput_GVL.Digital_Output[26], behaviour: TOGGLE
    ImageSwitcher (31,257 15x15), variable: InputOutput_GVL.Digital_Output[27], behaviour: TOGGLE
    ImageSwitcher (31,278 15x15), variable: InputOutput_GVL.Digital_Output[28], behaviour: TOGGLE
    ImageSwitcher (31,299 15x15), variable: InputOutput_GVL.Digital_Output[29], behaviour: TOGGLE
    ImageSwitcher (31,320 15x15), variable: InputOutput_GVL.Digital_Output[30], behaviour: TOGGLE
    ImageSwitcher (31,342 15x15), variable: InputOutput_GVL.Digital_Output[31], behaviour: TOGGLE
    ImageSwitcher (31,363 15x15), variable: InputOutput_GVL.Digital_Output[32], behaviour: TOGGLE
    Button (769,-1 30x30), image: VisuSymbols.Symbols.Wrong
        OnMouseClick: CloseDialog Dialog=P2_DO2, Result=OK, NumpadKeypadSet=True
END_VISUALIZATION

// ---- VISUs/PLC Status/P2 - Panel Outfeed/P2_DO3.TcVIS
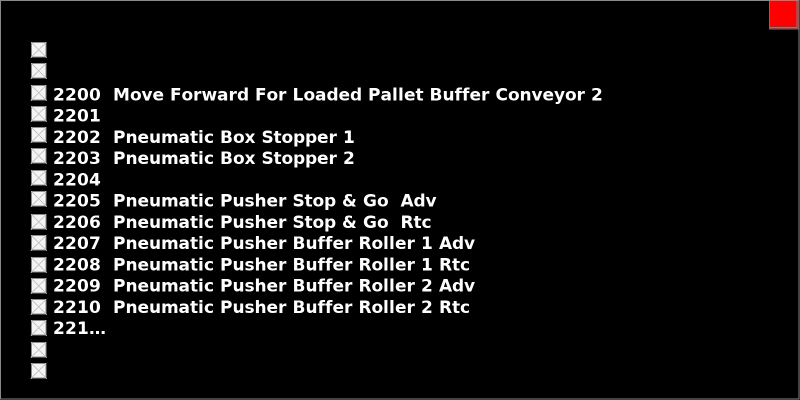
VISUALIZATION P2_DO3  // 800x400, background image 
    ImageSwitcher (31,42 15x15), variable: InputOutput_GVL.Digital_Output[33], behaviour: TOGGLE
    Label (50,16 625x391), "2200 Move Forward For Loaded Pallet Buffer Conveyor 2 2201 2202 Pneumatic Box Stopper 1 2203 Pneumatic Box Stopper 2 2204 2205 Pneumatic Pusher Stop & Go Adv 2206 Pneumatic Pusher Stop & Go Rtc 2207 Pneumatic Pusher Buffer Roller 1 Adv 2208 Pneumatic Pusher Buffer Roller 1 Rtc 2209 Pneumatic Pusher Buffer Roller 2 Adv 2210 Pneumatic Pusher Buffer Roller 2 Rtc 2211 2212 Interlock Status Infeed Modullar Busy 2213 Release Brake Motor Right Angle Lifter 2214 Interlock Request Pallet to Infeed Dispenser 2215 Interlock Request Pallet to Conveyor Outfeed Existing"
    ImageSwitcher (31,63 15x15), variable: InputOutput_GVL.Digital_Output[34], behaviour: TOGGLE
    ImageSwitcher (31,85 15x15), variable: InputOutput_GVL.Digital_Output[35], behaviour: TOGGLE
    ImageSwitcher (31,106 15x15), variable: InputOutput_GVL.Digital_Output[36], behaviour: TOGGLE
    ImageSwitcher (31,127 15x15), variable: InputOutput_GVL.Digital_Output[37], behaviour: TOGGLE
    ImageSwitcher (31,148 15x15), variable: InputOutput_GVL.Digital_Output[38], behaviour: TOGGLE
    ImageSwitcher (31,170 15x15), variable: InputOutput_GVL.Digital_Output[39], behaviour: TOGGLE
    ImageSwitcher (31,191 15x15), variable: InputOutput_GVL.Digital_Output[40], behaviour: TOGGLE
    ImageSwitcher (31,214 15x15), variable: InputOutput_GVL.Digital_Output[41], behaviour: TOGGLE
    ImageSwitcher (31,235 15x15), variable: InputOutput_GVL.Digital_Output[42], behaviour: TOGGLE
    ImageSwitcher (31,257 15x15), variable: InputOutput_GVL.Digital_Output[43], behaviour: TOGGLE
    ImageSwitcher (31,278 15x15), variable: InputOutput_GVL.Digital_Output[44], behaviour: TOGGLE
    ImageSwitcher (31,299 15x15), variable: InputOutput_GVL.Digital_Output[45], behaviour: TOGGLE
    ImageSwitcher (31,320 15x15), variable: InputOutput_GVL.Digital_Output[46], behaviour: TOGGLE
    ImageSwitcher (31,342 15x15), variable: InputOutput_GVL.Digital_Output[47], behaviour: TOGGLE
    ImageSwitcher (31,363 15x15), variable: InputOutput_GVL.Digital_Output[48], behaviour: TOGGLE
    Button (769,-1 30x30), image: VisuSymbols.Symbols.Wrong
        OnMouseClick: CloseDialog Dialog=P2_DO3, Result=OK, NumpadKeypadSet=True
END_VISUALIZATION

// ---- VISUs/PLC Status/P2 - Panel Outfeed/P2_DO4.TcVIS
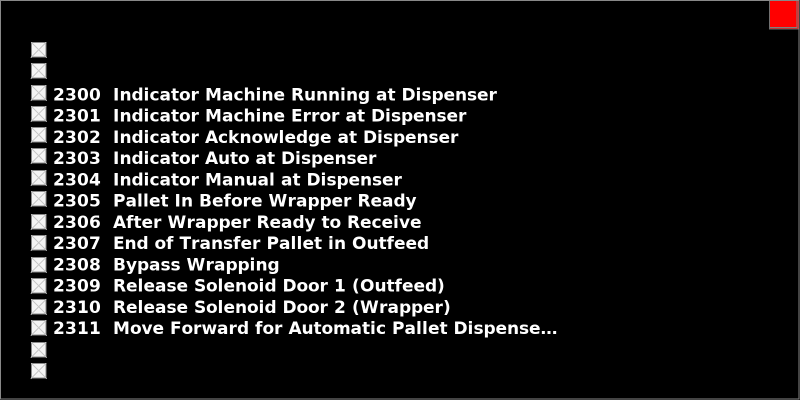
VISUALIZATION P2_DO4  // 800x400, background image 
    ImageSwitcher (31,42 15x15), variable: InputOutput_GVL.Digital_Output[49], behaviour: TOGGLE
    Label (50,16 625x391), "2300 Indicator Machine Running at Dispenser 2301 Indicator Machine Error at Dispenser 2302 Indicator Acknowledge at Dispenser 2303 Indicator Auto at Dispenser 2304 Indicator Manual at Dispenser 2305 Pallet In Before Wrapper Ready 2306 After Wrapper Ready to Receive 2307 End of Transfer Pallet in Outfeed 2308 Bypass Wrapping 2309 Release Solenoid Door 1 (Outfeed) 2310 Release Solenoid Door 2 (Wrapper) 2311 Move Forward for Automatic Pallet Dispenser 2312 Pneumatic Vertical Up 2313 Pneumatic Vertical Down 2314 Pneumatic Horizontal Rectract 2315 Pneumatic Horizontal Advanced"
    ImageSwitcher (31,63 15x15), variable: InputOutput_GVL.Digital_Output[50], behaviour: TOGGLE
    ImageSwitcher (31,85 15x15), variable: InputOutput_GVL.Digital_Output[51], behaviour: TOGGLE
    ImageSwitcher (31,106 15x15), variable: InputOutput_GVL.Digital_Output[52], behaviour: TOGGLE
    ImageSwitcher (31,127 15x15), variable: InputOutput_GVL.Digital_Output[53], behaviour: TOGGLE
    ImageSwitcher (31,148 15x15), variable: InputOutput_GVL.Digital_Output[54], behaviour: TOGGLE
    ImageSwitcher (31,170 15x15), variable: InputOutput_GVL.Digital_Output[55], behaviour: TOGGLE
    ImageSwitcher (31,191 15x15), variable: InputOutput_GVL.Digital_Output[56], behaviour: TOGGLE
    ImageSwitcher (31,214 15x15), variable: InputOutput_GVL.Digital_Output[57], behaviour: TOGGLE
    ImageSwitcher (31,235 15x15), variable: InputOutput_GVL.Digital_Output[58], behaviour: TOGGLE
    ImageSwitcher (31,257 15x15), variable: InputOutput_GVL.Digital_Output[59], behaviour: TOGGLE
    ImageSwitcher (31,278 15x15), variable: InputOutput_GVL.Digital_Output[60], behaviour: TOGGLE
    ImageSwitcher (31,299 15x15), variable: InputOutput_GVL.Digital_Output[61], behaviour: TOGGLE
    ImageSwitcher (31,320 15x15), variable: InputOutput_GVL.Digital_Output[62], behaviour: TOGGLE
    ImageSwitcher (31,342 15x15), variable: InputOutput_GVL.Digital_Output[63], behaviour: TOGGLE
    ImageSwitcher (31,363 15x15), variable: InputOutput_GVL.Digital_Output[64], behaviour: TOGGLE
    Button (769,-1 30x30), image: VisuSymbols.Symbols.Wrong
        OnMouseClick: CloseDialog Dialog=P2_DO4, Result=OK, NumpadKeypadSet=True
END_VISUALIZATION

// ---- VISUs/PLC Status/P3 - Panel Shuttle/P3_DI1.TcVIS
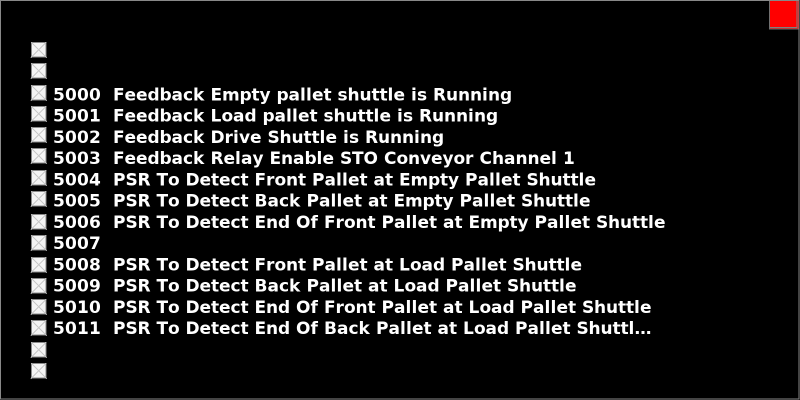
VISUALIZATION P3_DI1  // 800x400, background image 
    ImageSwitcher (31,42 15x15), variable: InputOutput_GVL.Digital_Input[113], behaviour: TOGGLE
    Label (50,16 706x391), "5000 Feedback Empty pallet shuttle is Running 5001 Feedback Load pallet shuttle is Running 5002 Feedback Drive Shuttle is Running 5003 Feedback Relay Enable STO Conveyor Channel 1 5004 PSR To Detect Front Pallet at Empty Pallet Shuttle 5005 PSR To Detect Back Pallet at Empty Pallet Shuttle 5006 PSR To Detect End Of Front Pallet at Empty Pallet Shuttle 5007 5008 PSR To Detect Front Pallet at Load Pallet Shuttle 5009 PSR To Detect Back Pallet at Load Pallet Shuttle 5010 PSR To Detect End Of Front Pallet at Load Pallet Shuttle 5011 PSR To Detect End Of Back Pallet at Load Pallet Shuttle 5012 Limit Switch To Detect Left Limit Area 5013 Limit Switch To Detect Right Limit Area 5014 PRX to Detect Left Limit Area 5015 PRX to Detect Right Limit Area"
    ImageSwitcher (31,63 15x15), variable: InputOutput_GVL.Digital_Input[114], behaviour: TOGGLE
    ImageSwitcher (31,85 15x15), variable: InputOutput_GVL.Digital_Input[115], behaviour: TOGGLE
    ImageSwitcher (31,106 15x15), variable: InputOutput_GVL.Digital_Input[116], behaviour: TOGGLE
    ImageSwitcher (31,127 15x15), variable: InputOutput_GVL.Digital_Input[117], behaviour: TOGGLE
    ImageSwitcher (31,148 15x15), variable: InputOutput_GVL.Digital_Input[118], behaviour: TOGGLE
    ImageSwitcher (31,170 15x15), variable: InputOutput_GVL.Digital_Input[119], behaviour: TOGGLE
    ImageSwitcher (31,191 15x15), variable: InputOutput_GVL.Digital_Input[120], behaviour: TOGGLE
    ImageSwitcher (31,214 15x15), variable: InputOutput_GVL.Digital_Input[121], behaviour: TOGGLE
    ImageSwitcher (31,235 15x15), variable: InputOutput_GVL.Digital_Input[122], behaviour: TOGGLE
    ImageSwitcher (31,257 15x15), variable: InputOutput_GVL.Digital_Input[123], behaviour: TOGGLE
    ImageSwitcher (31,278 15x15), variable: InputOutput_GVL.Digital_Input[124], behaviour: TOGGLE
    ImageSwitcher (31,299 15x15), variable: InputOutput_GVL.Digital_Input[125], behaviour: TOGGLE
    ImageSwitcher (31,320 15x15), variable: InputOutput_GVL.Digital_Input[126], behaviour: TOGGLE
    ImageSwitcher (31,342 15x15), variable: InputOutput_GVL.Digital_Input[127], behaviour: TOGGLE
    ImageSwitcher (31,363 15x15), variable: InputOutput_GVL.Digital_Input[128], behaviour: TOGGLE
    Button (769,-1 30x30), image: VisuSymbols.Symbols.Wrong
        OnMouseClick: CloseDialog Dialog=P3_DI1, Result=OK, NumpadKeypadSet=True
END_VISUALIZATION

// ---- VISUs/PLC Status/P3 - Panel Shuttle/P3_DO1.TcVIS
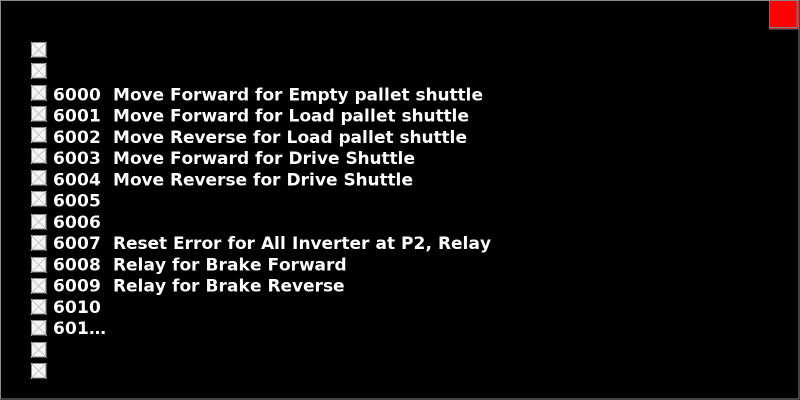
VISUALIZATION P3_DO1  // 800x400, background image 
    ImageSwitcher (31,42 15x15), variable: InputOutput_GVL.Digital_Output[65], behaviour: TOGGLE
    Label (50,16 625x391), "6000 Move Forward for Empty pallet shuttle 6001 Move Forward for Load pallet shuttle 6002 Move Reverse for Load pallet shuttle 6003 Move Forward for Drive Shuttle 6004 Move Reverse for Drive Shuttle 6005 6006 6007 Reset Error for All Inverter at P2, Relay 6008 Relay for Brake Forward 6009 Relay for Brake Reverse 6010 6011 6012 6013 6014 6015"
    ImageSwitcher (31,63 15x15), variable: InputOutput_GVL.Digital_Output[66], behaviour: TOGGLE
    ImageSwitcher (31,85 15x15), variable: InputOutput_GVL.Digital_Output[67], behaviour: TOGGLE
    ImageSwitcher (31,106 15x15), variable: InputOutput_GVL.Digital_Output[68], behaviour: TOGGLE
    ImageSwitcher (31,127 15x15), variable: InputOutput_GVL.Digital_Output[69], behaviour: TOGGLE
    ImageSwitcher (31,148 15x15), variable: InputOutput_GVL.Digital_Output[70], behaviour: TOGGLE
    ImageSwitcher (31,170 15x15), variable: InputOutput_GVL.Digital_Output[71], behaviour: TOGGLE
    ImageSwitcher (31,191 15x15), variable: InputOutput_GVL.Digital_Output[72], behaviour: TOGGLE
    ImageSwitcher (31,214 15x15), variable: InputOutput_GVL.Digital_Output[73], behaviour: TOGGLE
    ImageSwitcher (31,235 15x15), variable: InputOutput_GVL.Digital_Output[74], behaviour: TOGGLE
    ImageSwitcher (31,257 15x15), variable: InputOutput_GVL.Digital_Output[75], behaviour: TOGGLE
    ImageSwitcher (31,278 15x15), variable: InputOutput_GVL.Digital_Output[76], behaviour: TOGGLE
    ImageSwitcher (31,299 15x15), variable: InputOutput_GVL.Digital_Output[77], behaviour: TOGGLE
    ImageSwitcher (31,320 15x15), variable: InputOutput_GVL.Digital_Output[78], behaviour: TOGGLE
    ImageSwitcher (31,342 15x15), variable: InputOutput_GVL.Digital_Output[79], behaviour: TOGGLE
    ImageSwitcher (31,363 15x15), variable: InputOutput_GVL.Digital_Output[80], behaviour: TOGGLE
    Button (769,-1 30x30), image: VisuSymbols.Symbols.Wrong
        OnMouseClick: CloseDialog Dialog=P3_DO1, Result=OK, NumpadKeypadSet=True
END_VISUALIZATION

// ---- VISUs/PLC Status/SeqStatus.TcVIS
